// TwinCAT 3 PLC project Untitled1
// ProgramVersion: 3.1.4022.7
// libraries:
//   Tc2_Standard, * (Beckhoff Automation GmbH)
//   Tc2_System, * (Beckhoff Automation GmbH)
//   Tc3_Module, * (Beckhoff Automation GmbH)
// project tree:
//   / PlcTask.TcTTO
//   POUs/ alg_s_Dinitialized.TcPOU, alg_s_Hinitialized.TcPOU, alg_a_Dstartled.TcPOU (not stored), alg_a_Dresetled.TcPOU (not stored), alg_a_DledQ1.TcPOU (not stored), alg_a_DledQ2.TcPOU (not stored), alg_a_pusher1.TcPOU (not stored), alg_a_pusher2.TcPOU (not stored), alg_a_pusher3.TcPOU (not stored), alg_a_Hstartled.TcPOU (not stored), alg_a_Hresetled.TcPOU (not stored), alg_a_HledQ1.TcPOU (not stored), alg_a_HledQ2.TcPOU (not stored), alg_a_x2distributing.TcPOU (not stored), alg_a_x2testing.TcPOU (not stored), alg_a_zdown.TcPOU (not stored), alg_a_gripperclose.TcPOU (not stored), alg_a_transfer2pickpos.TcPOU (not stored), alg_a_transfer2droppos.TcPOU (not stored), alg_a_vacuum.TcPOU (not stored), alg_a_ejectpulse.TcPOU (not stored), alg_a_handlingready.TcPOU (not stored), alg_M_Distributing_a_Dstopled.TcPOU (not stored), alg_M_Distributing_a_Dstartled.TcPOU (not stored), alg_M_Distributing_a_Dresetled.TcPOU (not stored), alg_M_Distributing_pickpos.TcPOU (not stored), makeArray0.TcPOU (not stored), alg_M_Distributing_atpos.TcPOU (not stored), makeArray1.TcPOU (not stored), derivcvar_M_Distributing_t.TcPOU (not stored), ifExprFunc1.TcPOU (not stored), derivcvar_M_HardwareMap_t.TcPOU, MAIN.TcPOU, projArray0.TcPOU (not stored), normProjIdx.TcPOU (not stored), projArray1.TcPOU (not stored)
//   DUTs/ STATE.TcDUT, enum_E.TcDUT
//   GVLs/ INPUTS.TcGVL, TIMERS.TcGVL
// real-time tasks:
//   TASK PlcTask: cycle T#10ms, priority 20, ADS port 350
// I/O:
//   DEVICE Device 2 (EtherCAT), AmsNetId 192.168.1.11.3.1
//     Term 1 (EK1100) [EK1100 EtherCAT Coupler (2A E-Bus)]
//       Term 2 (EL2828) [EL2828 8Ch. Dig. Output 24V, 2A]
//       Term 3 (EL1008) [EL1008 8Ch. Dig. Input 24V, 3ms]
//       Term 4 (EL2024) [EL2024 4Ch. Dig. Output 24V, 2A]
//       Term 5 (EL1008) [EL1008 8Ch. Dig. Input 24V, 3ms]
//       Term 6 (EL2024) [EL2024 4Ch. Dig. Output 24V, 2A]
//       Term 7 (EL1008) [EL1008 8Ch. Dig. Input 24V, 3ms]
//       Term 16 (EL9011) [EL9011 End Terminal]
//     Term 8 (EK1100) [EK1100 EtherCAT Coupler (2A E-Bus)]
//       Term 9 (EL2828) [EL2828 8Ch. Dig. Output 24V, 2A]
//       Term 10 (EL1008) [EL1008 8Ch. Dig. Input 24V, 3ms]
//       Term 11 (EL2024) [EL2024 4Ch. Dig. Output 24V, 2A]
//       Term 12 (EL2024) [EL2024 4Ch. Dig. Output 24V, 2A]
//       Term 13 (EL1008) [EL1008 8Ch. Dig. Input 24V, 3ms]
//       Term 14 (EL2004) [EL2004 4Ch. Dig. Output 24V, 0.5A]
//       Term 15 (EL1008) [EL1008 8Ch. Dig. Input 24V, 3ms]
//       Term 17 (EL9011) [EL9011 End Terminal]
// variable links:
//   Untitled1/Untitled1 Instance <-> Device 2 (EtherCAT)/Term 1 (EK1100)/Term 2 (EL2828)
//     PlcTask Outputs/MAIN.state0.dvar_M_HardwareMap_out_a_DledQ1 <-> Channel 3/Output
//     PlcTask Outputs/MAIN.state0.dvar_M_HardwareMap_out_a_DledQ2 <-> Channel 4/Output
//     PlcTask Outputs/MAIN.state0.dvar_M_HardwareMap_out_a_Dout{4..7} <-> Channel {5..8}/Output  (4 links)
//     PlcTask Outputs/MAIN.state0.dvar_M_HardwareMap_out_a_Dresetled <-> Channel 2/Output
//     PlcTask Outputs/MAIN.state0.dvar_M_HardwareMap_out_a_Dstartled <-> Channel 1/Output
//   Untitled1/Untitled1 Instance <-> Device 2 (EtherCAT)/Term 1 (EK1100)/Term 3 (EL1008)
//     PlcTask Inputs/INPUTS.ivar_s_Dautoswitch <-> Channel 3/Input
//     PlcTask Inputs/INPUTS.ivar_s_Din{4..7} <-> Channel {5..8}/Input  (4 links)
//     PlcTask Inputs/INPUTS.ivar_s_Dresetbutton <-> Channel 4/Input
//     PlcTask Inputs/INPUTS.ivar_s_Dstartbutton <-> Channel 1/Input
//     PlcTask Inputs/INPUTS.ivar_s_Dstopbutton <-> Channel 2/Input
//   Untitled1/Untitled1 Instance <-> Device 2 (EtherCAT)/Term 1 (EK1100)/Term 4 (EL2024)
//     PlcTask Outputs/MAIN.state0.dvar_M_HardwareMap_out_a_pusher1 <-> Channel 1/Output
//     PlcTask Outputs/MAIN.state0.dvar_M_HardwareMap_out_a_pusher2 <-> Channel 2/Output
//     PlcTask Outputs/MAIN.state0.dvar_M_HardwareMap_out_a_pusher3 <-> Channel 3/Output
//   Untitled1/Untitled1 Instance <-> Device 2 (EtherCAT)/Term 1 (EK1100)/Term 5 (EL1008)
//     PlcTask Inputs/INPUTS.ivar_s_product1 <-> Channel 4/Input
//     PlcTask Inputs/INPUTS.ivar_s_product2 <-> Channel 8/Input
//     PlcTask Inputs/INPUTS.ivar_s_pusher1_in <-> Channel 1/Input
//     PlcTask Inputs/INPUTS.ivar_s_pusher2_in <-> Channel 5/Input
//     PlcTask Inputs/INPUTS.ivar_s_pusher1_out <-> Channel 2/Input
//     PlcTask Inputs/INPUTS.ivar_s_pusher2_out <-> Channel 6/Input
//     PlcTask Inputs/INPUTS.ivar_s_stack1filled <-> Channel 3/Input
//     PlcTask Inputs/INPUTS.ivar_s_stack2filled <-> Channel 7/Input
//   Untitled1/Untitled1 Instance <-> Device 2 (EtherCAT)/Term 1 (EK1100)/Term 7 (EL1008)
//     PlcTask Inputs/INPUTS.ivar_s_handlingbusy <-> Channel 8/Input
//     PlcTask Inputs/INPUTS.ivar_s_product3 <-> Channel 4/Input
//     PlcTask Inputs/INPUTS.ivar_s_pusher3_in <-> Channel 1/Input
//     PlcTask Inputs/INPUTS.ivar_s_pusher3_out <-> Channel 2/Input
//     PlcTask Inputs/INPUTS.ivar_s_stack3filled <-> Channel 3/Input
//   Untitled1/Untitled1 Instance <-> Device 2 (EtherCAT)/Term 8 (EK1100)/Term 10 (EL1008)
//     PlcTask Inputs/INPUTS.ivar_s_Hautoswitch <-> Channel 3/Input
//     PlcTask Inputs/INPUTS.ivar_s_Hin{4..7} <-> Channel {5..8}/Input  (4 links)
//     PlcTask Inputs/INPUTS.ivar_s_Hresetbutton <-> Channel 4/Input
//     PlcTask Inputs/INPUTS.ivar_s_Hstartbutton <-> Channel 1/Input
//     PlcTask Inputs/INPUTS.ivar_s_Hstopbutton <-> Channel 2/Input
//   Untitled1/Untitled1 Instance <-> Device 2 (EtherCAT)/Term 8 (EK1100)/Term 11 (EL2024)
//     PlcTask Outputs/MAIN.state0.dvar_M_HardwareMap_out_a_gripperclose <-> Channel 4/Output
//     PlcTask Outputs/MAIN.state0.dvar_M_HardwareMap_out_a_x2distributing <-> Channel 1/Output
//     PlcTask Outputs/MAIN.state0.dvar_M_HardwareMap_out_a_x2testing <-> Channel 2/Output
//     PlcTask Outputs/MAIN.state0.dvar_M_HardwareMap_out_a_zdown <-> Channel 3/Output
//   Untitled1/Untitled1 Instance <-> Device 2 (EtherCAT)/Term 8 (EK1100)/Term 12 (EL2024)
//     PlcTask Outputs/MAIN.state0.dvar_M_HardwareMap_out_a_ejectpulse <-> Channel 4/Output
//     PlcTask Outputs/MAIN.state0.dvar_M_HardwareMap_out_a_transfer2droppos <-> Channel 2/Output
//     PlcTask Outputs/MAIN.state0.dvar_M_HardwareMap_out_a_transfer2pickpos <-> Channel 1/Output
//     PlcTask Outputs/MAIN.state0.dvar_M_HardwareMap_out_a_vacuum <-> Channel 3/Output
//   Untitled1/Untitled1 Instance <-> Device 2 (EtherCAT)/Term 8 (EK1100)/Term 13 (EL1008)
//     PlcTask Inputs/INPUTS.ivar_s_xpos_at1 <-> Channel 4/Input
//     PlcTask Inputs/INPUTS.ivar_s_xpos_at2 <-> Channel 5/Input
//     PlcTask Inputs/INPUTS.ivar_s_xpos_at3 <-> Channel 6/Input
//     PlcTask Inputs/INPUTS.ivar_s_xpos_atdrop <-> Channel 7/Input
//     PlcTask Inputs/INPUTS.ivar_s_zpos_atup <-> Channel 8/Input
//   Untitled1/Untitled1 Instance <-> Device 2 (EtherCAT)/Term 8 (EK1100)/Term 14 (EL2004)
//     PlcTask Outputs/MAIN.state0.dvar_M_HardwareMap_out_a_handlingready <-> Channel 4/Output
//   Untitled1/Untitled1 Instance <-> Device 2 (EtherCAT)/Term 8 (EK1100)/Term 15 (EL1008)
//     PlcTask Inputs/INPUTS.ivar_s_gripper <-> Channel 2/Input
//     PlcTask Inputs/INPUTS.ivar_s_product4 <-> Channel 7/Input
//     PlcTask Inputs/INPUTS.ivar_s_testingbusy <-> Channel 8/Input
//     PlcTask Inputs/INPUTS.ivar_s_transfer_atdrop <-> Channel 4/Input
//     PlcTask Inputs/INPUTS.ivar_s_transfer_athalfway <-> Channel 5/Input
//     PlcTask Inputs/INPUTS.ivar_s_transfer_atpickup <-> Channel 3/Input
//     PlcTask Inputs/INPUTS.ivar_s_vacuum <-> Channel 6/Input
//     PlcTask Inputs/INPUTS.ivar_s_zpos_atdown <-> Channel 1/Input
//   Untitled1/Untitled1 Instance <-> Device 2 (EtherCAT)/Term 8 (EK1100)/Term 9 (EL2828)
//     PlcTask Outputs/MAIN.state0.dvar_M_HardwareMap_out_a_HledQ1 <-> Channel 3/Output
//     PlcTask Outputs/MAIN.state0.dvar_M_HardwareMap_out_a_HledQ2 <-> Channel 4/Output
//     PlcTask Outputs/MAIN.state0.dvar_M_HardwareMap_out_a_Hout{4..7} <-> Channel {5..8}/Output  (4 links)
//     PlcTask Outputs/MAIN.state0.dvar_M_HardwareMap_out_a_Hresetled <-> Channel 2/Output
//     PlcTask Outputs/MAIN.state0.dvar_M_HardwareMap_out_a_Hstartled <-> Channel 1/Output

CONFIGURATION Untitled1
    RESOURCE PLC ON TwinCAT3
        TASK PlcTask(INTERVAL := T#10ms, PRIORITY := 20);
        PROGRAM MAIN WITH PlcTask : MAIN;
    END_RESOURCE
END_CONFIGURATION

// ---- DUTs/STATE.TcDUT
TYPE STATE:
    STRUCT
        curTime: LREAL;
        dvar_M_Distributing_a_x2distributing AT %Q*: BOOL;
        dvar_M_Distributing_a_zdown AT %Q*: BOOL;
        dvar_M_Distributing_a_gripperclose AT %Q*: BOOL;
        dvar_M_Distributing_a_x2testing AT %Q*: BOOL;
        dvar_M_Distributing_i AT %Q*: DINT;
        cvar_M_Distributing_t AT %Q*: LREAL;
        dvar_M_Distributing AT %Q*: enum_E;
        dvar_M_HardwareMap_out_a_Dstartled AT %Q*: BOOL;
        dvar_M_HardwareMap_out_a_Dresetled AT %Q*: BOOL;
        dvar_M_HardwareMap_out_a_DledQ1 AT %Q*: BOOL;
        dvar_M_HardwareMap_out_a_DledQ2 AT %Q*: BOOL;
        dvar_M_HardwareMap_out_a_Dout4 AT %Q*: BOOL;
        dvar_M_HardwareMap_out_a_Dout5 AT %Q*: BOOL;
        dvar_M_HardwareMap_out_a_Dout6 AT %Q*: BOOL;
        dvar_M_HardwareMap_out_a_Dout7 AT %Q*: BOOL;
        dvar_M_HardwareMap_out_a_pusher1 AT %Q*: BOOL;
        dvar_M_HardwareMap_out_a_pusher2 AT %Q*: BOOL;
        dvar_M_HardwareMap_out_a_pusher3 AT %Q*: BOOL;
        dvar_M_HardwareMap_out_a_Hstartled AT %Q*: BOOL;
        dvar_M_HardwareMap_out_a_Hresetled AT %Q*: BOOL;
        dvar_M_HardwareMap_out_a_HledQ1 AT %Q*: BOOL;
        dvar_M_HardwareMap_out_a_HledQ2 AT %Q*: BOOL;
        dvar_M_HardwareMap_out_a_Hout4 AT %Q*: BOOL;
        dvar_M_HardwareMap_out_a_Hout5 AT %Q*: BOOL;
        dvar_M_HardwareMap_out_a_Hout6 AT %Q*: BOOL;
        dvar_M_HardwareMap_out_a_Hout7 AT %Q*: BOOL;
        dvar_M_HardwareMap_out_a_x2distributing AT %Q*: BOOL;
        dvar_M_HardwareMap_out_a_x2testing AT %Q*: BOOL;
        dvar_M_HardwareMap_out_a_zdown AT %Q*: BOOL;
        dvar_M_HardwareMap_out_a_gripperclose AT %Q*: BOOL;
        dvar_M_HardwareMap_out_a_transfer2pickpos AT %Q*: BOOL;
        dvar_M_HardwareMap_out_a_transfer2droppos AT %Q*: BOOL;
        dvar_M_HardwareMap_out_a_vacuum AT %Q*: BOOL;
        dvar_M_HardwareMap_out_a_ejectpulse AT %Q*: BOOL;
        dvar_M_HardwareMap_out_a_handlingready AT %Q*: BOOL;
        dvar_M_HardwareMap_init_err_sen_idx AT %Q*: DINT;
        dvar_M_HardwareMap_init_err_led_idx AT %Q*: DINT;
        cvar_M_HardwareMap_t AT %Q*: LREAL;
        dvar_M_HardwareMap AT %Q*: enum_E;
        dvar_M_inventory1_a_pusher1 AT %Q*: BOOL;
        dvar_M_inventory1 AT %Q*: enum_E;
        dvar_M_inventory2_a_pusher2 AT %Q*: BOOL;
        dvar_M_inventory2 AT %Q*: enum_E;
        dvar_M_inventory3_a_pusher3 AT %Q*: BOOL;
        dvar_M_inventory3 AT %Q*: enum_E;
        dvar_M_vacuum_a_transfer2pickpos AT %Q*: BOOL;
        dvar_M_vacuum_a_transfer2droppos AT %Q*: BOOL;
        dvar_M_vacuum_a_vacuum AT %Q*: BOOL;
        dvar_M_vacuum_a_ejectpulse AT %Q*: BOOL;
        dvar_M_vacuum AT %Q*: enum_E;
    END_STRUCT
END_TYPE

// ---- DUTs/enum_E.TcDUT
TYPE enum_E:
    (elit_clear_vacuum, elit_down, elit_droppoint, elit_finished, elit_goback, elit_going, elit_gopickup, elit_goup, elit_init0, elit_init1, elit_init2, elit_init3, elit_init4, elit_init5, elit_init6, elit_init7, elit_init8, elit_init9, elit_init_error, elit_init_ok, elit_init_sensor_check, elit_initialized, elit_key, elit_movetopickup, elit_pauze_left, elit_pickupvac, elit_reset, elit_reset_button, elit_reset_down, elit_reset_place, elit_rest, elit_starting, elit_stop, elit_testingdrop, elit_wait_start, elit_wait_vacuum);
END_TYPE

// ---- GVLs/INPUTS.TcGVL
VAR_GLOBAL // INPUTS
    ivar_s_Dstartbutton AT %I*: BOOL;
    ivar_s_Dstopbutton AT %I*: BOOL;
    ivar_s_Dresetbutton AT %I*: BOOL;
    ivar_s_Dautoswitch AT %I*: BOOL;
    ivar_s_pusher1_in AT %I*: BOOL;
    ivar_s_pusher1_out AT %I*: BOOL;
    ivar_s_stack1filled AT %I*: BOOL;
    ivar_s_product1 AT %I*: BOOL;
    ivar_s_pusher2_in AT %I*: BOOL;
    ivar_s_pusher2_out AT %I*: BOOL;
    ivar_s_stack2filled AT %I*: BOOL;
    ivar_s_product2 AT %I*: BOOL;
    ivar_s_pusher3_in AT %I*: BOOL;
    ivar_s_pusher3_out AT %I*: BOOL;
    ivar_s_stack3filled AT %I*: BOOL;
    ivar_s_product3 AT %I*: BOOL;
    ivar_s_handlingbusy AT %I*: BOOL;
    ivar_s_Hstartbutton AT %I*: BOOL;
    ivar_s_Hstopbutton AT %I*: BOOL;
    ivar_s_Hresetbutton AT %I*: BOOL;
    ivar_s_Hautoswitch AT %I*: BOOL;
    ivar_s_xpos_at1 AT %I*: BOOL;
    ivar_s_xpos_at2 AT %I*: BOOL;
    ivar_s_xpos_at3 AT %I*: BOOL;
    ivar_s_xpos_atdrop AT %I*: BOOL;
    ivar_s_zpos_atup AT %I*: BOOL;
    ivar_s_zpos_atdown AT %I*: BOOL;
    ivar_s_gripper AT %I*: BOOL;
    ivar_s_transfer_atpickup AT %I*: BOOL;
    ivar_s_transfer_atdrop AT %I*: BOOL;
    ivar_s_transfer_athalfway AT %I*: BOOL;
    ivar_s_vacuum AT %I*: BOOL;
    ivar_s_product4 AT %I*: BOOL;
    ivar_s_testingbusy AT %I*: BOOL;
    ivar_s_Din4 AT %I*: BOOL;
    ivar_s_Din5 AT %I*: BOOL;
    ivar_s_Din6 AT %I*: BOOL;
    ivar_s_Din7 AT %I*: BOOL;
    ivar_s_Hin4 AT %I*: BOOL;
    ivar_s_Hin5 AT %I*: BOOL;
    ivar_s_Hin6 AT %I*: BOOL;
    ivar_s_Hin7 AT %I*: BOOL;
    ivar_a_Dout4 AT %I*: BOOL;
    ivar_a_Dout5 AT %I*: BOOL;
    ivar_a_Dout6 AT %I*: BOOL;
    ivar_a_Dout7 AT %I*: BOOL;
    ivar_a_Hout4 AT %I*: BOOL;
    ivar_a_Hout5 AT %I*: BOOL;
    ivar_a_Hout6 AT %I*: BOOL;
    ivar_a_Hout7 AT %I*: BOOL;
END_VAR

// ---- GVLs/TIMERS.TcGVL
VAR_GLOBAL // TIMERS
    timer0: TON;
    timer1: TON;
    curTimer: INT := 0;
END_VAR

// ---- POUs/MAIN.TcPOU
PROGRAM MAIN
VAR_OUTPUT
    timerValue0: TIME;
    timerValue1: TIME;
END_VAR
VAR
    cnt: LINT;
    first: BOOL := TRUE;
    curTimerValue: TIME;
    state0: STATE;
    curTime: LREAL;
    loopsKilled: LINT;
END_VAR
VAR_TEMP
    lastTimerValue: TIME;
    curDeltaTime: TIME;
    curDeltaSecs: LREAL;
    state1: STATE;
    progress: BOOL;
    loopCount: INT;
    b1: BOOL;
    b2: BOOL;
END_VAR


// Handle 'time' and cycle time.
cnt := cnt + 1;

timer0(IN := curTimer = 0, PT := T#1D);
timer1(IN := curTimer = 1, PT := T#1D);
timerValue0 := timer0.ET;
timerValue1 := timer1.ET;

lastTimerValue := curTimerValue;
IF curTimer = 0 THEN
    curTimerValue := timerValue0;
ELSE
    curTimerValue := timerValue1;
END_IF;
curDeltaTime := curTimerValue - lastTimerValue;
curDeltaSecs := TIME_TO_LREAL(curDeltaTime) / 1000;
curTime := curTime + curDeltaSecs;

IF cnt MOD 10 = 0 THEN
    curTimer := 1 - curTimer;
    curTimerValue := T#0S;
    timer0(IN := curTimer = 0, PT := T#1D);
    timer1(IN := curTimer = 1, PT := T#1D);
    timerValue0 := timer0.ET;
    timerValue1 := timer1.ET;
END_IF;

IF first THEN
    first := FALSE;

    // Initialize state variables for initial state.
    state0.dvar_M_Distributing_a_x2distributing := FALSE;
    state0.dvar_M_Distributing_a_zdown := FALSE;
    state0.dvar_M_Distributing_a_gripperclose := FALSE;
    state0.dvar_M_Distributing_a_x2testing := FALSE;
    state0.dvar_M_Distributing_i := 0;
    state0.cvar_M_Distributing_t := 0.0;
    state0.dvar_M_Distributing := elit_init2;
    state0.dvar_M_HardwareMap_out_a_Dstartled := FALSE;
    state0.dvar_M_HardwareMap_out_a_Dresetled := FALSE;
    state0.dvar_M_HardwareMap_out_a_DledQ1 := TRUE;
    state0.dvar_M_HardwareMap_out_a_DledQ2 := TRUE;
    state0.dvar_M_HardwareMap_out_a_Dout4 := FALSE;
    state0.dvar_M_HardwareMap_out_a_Dout5 := FALSE;
    state0.dvar_M_HardwareMap_out_a_Dout6 := FALSE;
    state0.dvar_M_HardwareMap_out_a_Dout7 := FALSE;
    state0.dvar_M_HardwareMap_out_a_pusher1 := FALSE;
    state0.dvar_M_HardwareMap_out_a_pusher2 := FALSE;
    state0.dvar_M_HardwareMap_out_a_pusher3 := FALSE;
    state0.dvar_M_HardwareMap_out_a_Hstartled := FALSE;
    state0.dvar_M_HardwareMap_out_a_Hresetled := FALSE;
    state0.dvar_M_HardwareMap_out_a_HledQ1 := TRUE;
    state0.dvar_M_HardwareMap_out_a_HledQ2 := TRUE;
    state0.dvar_M_HardwareMap_out_a_Hout4 := FALSE;
    state0.dvar_M_HardwareMap_out_a_Hout5 := FALSE;
    state0.dvar_M_HardwareMap_out_a_Hout6 := FALSE;
    state0.dvar_M_HardwareMap_out_a_Hout7 := FALSE;
    state0.dvar_M_HardwareMap_out_a_x2distributing := TRUE;
    state0.dvar_M_HardwareMap_out_a_x2testing := TRUE;
    state0.dvar_M_HardwareMap_out_a_zdown := FALSE;
    state0.dvar_M_HardwareMap_out_a_gripperclose := FALSE;
    state0.dvar_M_HardwareMap_out_a_transfer2pickpos := FALSE;
    state0.dvar_M_HardwareMap_out_a_transfer2droppos := FALSE;
    state0.dvar_M_HardwareMap_out_a_vacuum := FALSE;
    state0.dvar_M_HardwareMap_out_a_ejectpulse := FALSE;
    state0.dvar_M_HardwareMap_out_a_handlingready := FALSE;
    state0.dvar_M_HardwareMap_init_err_sen_idx := -1;
    state0.dvar_M_HardwareMap_init_err_led_idx := 0;
    state0.cvar_M_HardwareMap_t := 0.0;
    state0.dvar_M_HardwareMap := elit_init0;
    state0.dvar_M_inventory1_a_pusher1 := FALSE;
    state0.dvar_M_inventory1 := elit_init2;
    state0.dvar_M_inventory2_a_pusher2 := FALSE;
    state0.dvar_M_inventory2 := elit_init2;
    state0.dvar_M_inventory3_a_pusher3 := FALSE;
    state0.dvar_M_inventory3 := elit_init2;
    state0.dvar_M_vacuum_a_transfer2pickpos := FALSE;
    state0.dvar_M_vacuum_a_transfer2droppos := FALSE;
    state0.dvar_M_vacuum_a_vacuum := FALSE;
    state0.dvar_M_vacuum_a_ejectpulse := FALSE;
    state0.dvar_M_vacuum := elit_init2;
ELSE
    // Update continuous variables for time delay.
    state1.cvar_M_Distributing_t := state0.cvar_M_Distributing_t + curDeltaSecs * derivcvar_M_Distributing_t(state0);
    state1.cvar_M_HardwareMap_t := state0.cvar_M_HardwareMap_t + curDeltaSecs * derivcvar_M_HardwareMap_t(state0);

    state0.curTime := curTime;
    state0.cvar_M_Distributing_t := state1.cvar_M_Distributing_t;
    state0.cvar_M_HardwareMap_t := state1.cvar_M_HardwareMap_t;
END_IF;

// Event loop.
WHILE TRUE DO
    progress := FALSE;

    // Event "M.inventory1_a".
    IF NOT progress THEN
        b1 := (state0.dvar_M_inventory1) = (elit_starting);
        b1 := b1 AND (ivar_s_pusher1_in);
        b1 := b1 AND (NOT(ivar_s_product1));
        IF b1 THEN
            progress := TRUE;
            state1 := state0;

            state1.dvar_M_inventory1_a_pusher1 := TRUE;
            state1.dvar_M_inventory1 := elit_going;

            state0 := state1;
        END_IF;
    END_IF;

    // Event "M.inventory1_b".
    IF NOT progress THEN
        b1 := (state0.dvar_M_inventory1) = (elit_starting);
        b1 := b1 AND (ivar_s_pusher1_out);
        b1 := b1 AND (ivar_s_stack1filled);
        b1 := b1 AND (state0.dvar_M_inventory1_a_pusher1);
        IF b1 THEN
            progress := TRUE;
            state1 := state0;

            state1.dvar_M_inventory1 := elit_going;

            state0 := state1;
        END_IF;
    END_IF;

    // Event "M.inventory1_c".
    IF NOT progress THEN
        b1 := (state0.dvar_M_inventory1) = (elit_starting);
        b1 := b1 AND (NOT(ivar_s_Dstopbutton));
        IF b1 THEN
            progress := TRUE;
            state1 := state0;

            state1.dvar_M_inventory1_a_pusher1 := FALSE;
            state1.dvar_M_inventory1 := elit_stop;

            state0 := state1;
        END_IF;
    END_IF;

    // Event "M.inventory1_d".
    IF NOT progress THEN
        b1 := (state0.dvar_M_inventory1) = (elit_going);
        b1 := b1 AND (ivar_s_pusher1_out);
        b1 := b1 AND (ivar_s_stack1filled);
        IF b1 THEN
            progress := TRUE;
            state1 := state0;

            state1.dvar_M_inventory1_a_pusher1 := FALSE;
            state1.dvar_M_inventory1 := elit_starting;

            state0 := state1;
        END_IF;
    END_IF;

    // Event "tau".
    IF NOT progress THEN
        b1 := (state0.dvar_M_Distributing) = (elit_init2);
        b1 := b1 AND (alg_s_Dinitialized(state0));
        IF b1 THEN
            progress := TRUE;
            state1 := state0;

            state1.dvar_M_Distributing := elit_wait_start;

            state0 := state1;
        END_IF;
    END_IF;

    // Event "tau".
    IF NOT progress THEN
        b1 := (state0.dvar_M_Distributing) = (elit_wait_start);
        b1 := b1 AND (ivar_s_Dstartbutton);
        IF b1 THEN
            progress := TRUE;
            state1 := state0;

            state1.dvar_M_Distributing := elit_droppoint;

            state0 := state1;
        END_IF;
    END_IF;

    // Event "tau".
    IF NOT progress THEN
        b1 := (state0.dvar_M_Distributing) = (elit_reset_button);
        b1 := b1 AND (NOT(ivar_s_Dstopbutton));
        IF b1 THEN
            progress := TRUE;
            state1 := state0;

            state1.dvar_M_Distributing_a_x2distributing := FALSE;
            state1.dvar_M_Distributing_a_x2testing := FALSE;
            state1.dvar_M_Distributing_a_zdown := FALSE;
            state1.dvar_M_Distributing := elit_stop;

            state0 := state1;
        END_IF;
    END_IF;

    // Event "tau".
    IF NOT progress THEN
        b1 := (state0.dvar_M_Distributing) = (elit_reset_button);
        b1 := b1 AND (ivar_s_gripper);
        b1 := b1 AND (ivar_s_xpos_at3);
        IF b1 THEN
            progress := TRUE;
            state1 := state0;

            state1.dvar_M_Distributing_a_zdown := FALSE;
            state1.dvar_M_Distributing_a_x2distributing := TRUE;
            state1.dvar_M_Distributing := elit_wait_vacuum;

            state0 := state1;
        END_IF;
    END_IF;

    // Event "tau".
    IF NOT progress THEN
        b1 := (state0.dvar_M_Distributing) = (elit_reset_button);
        b1 := b1 AND (ivar_s_gripper);
        b1 := b1 AND (ivar_s_xpos_atdrop);
        IF b1 THEN
            progress := TRUE;
            state1 := state0;

            state1.dvar_M_Distributing_a_zdown := FALSE;
            state1.dvar_M_Distributing_a_x2distributing := TRUE;
            state1.dvar_M_Distributing_a_x2testing := FALSE;
            state1.dvar_M_Distributing := elit_pauze_left;

            state0 := state1;
        END_IF;
    END_IF;

    // Event "tau".
    IF NOT progress THEN
        b1 := (state0.dvar_M_Distributing) = (elit_reset_button);
        b1 := b1 AND (NOT(ivar_s_gripper));
        b1 := b1 AND (ivar_s_xpos_at3);
        IF b1 THEN
            progress := TRUE;
            state1 := state0;

            state1.dvar_M_Distributing_a_zdown := FALSE;
            state1.dvar_M_Distributing_a_x2distributing := TRUE;
            state1.dvar_M_Distributing := elit_wait_vacuum;

            state0 := state1;
        END_IF;
    END_IF;

    // Event "tau".
    IF NOT progress THEN
        b1 := (state0.dvar_M_Distributing) = (elit_reset_button);
        b1 := b1 AND (NOT(ivar_s_gripper));
        b1 := b1 AND (ivar_s_xpos_atdrop);
        IF b1 THEN
            progress := TRUE;
            state1 := state0;

            state1.dvar_M_Distributing_a_zdown := FALSE;
            state1.dvar_M_Distributing_a_x2distributing := TRUE;
            state1.dvar_M_Distributing_a_x2testing := FALSE;
            state1.dvar_M_Distributing := elit_pauze_left;

            state0 := state1;
        END_IF;
    END_IF;

    // Event "tau".
    IF NOT progress THEN
        b1 := (state0.dvar_M_Distributing) = (elit_pauze_left);
        b1 := b1 AND (NOT(ivar_s_Dstopbutton));
        IF b1 THEN
            progress := TRUE;
            state1 := state0;

            state1.dvar_M_Distributing_a_x2distributing := FALSE;
            state1.dvar_M_Distributing_a_x2testing := FALSE;
            state1.dvar_M_Distributing_a_zdown := FALSE;
            state1.dvar_M_Distributing := elit_stop;

            state0 := state1;
        END_IF;
    END_IF;

    // Event "tau".
    IF NOT progress THEN
        b1 := (state0.dvar_M_Distributing) = (elit_pauze_left);
        b1 := b1 AND (NOT(ivar_s_gripper));
        b1 := b1 AND (ivar_s_xpos_at3);
        IF b1 THEN
            progress := TRUE;
            state1 := state0;

            state1.dvar_M_Distributing_a_zdown := FALSE;
            state1.dvar_M_Distributing_a_x2distributing := TRUE;
            state1.dvar_M_Distributing_a_x2testing := TRUE;
            state1.dvar_M_Distributing := elit_wait_vacuum;

            state0 := state1;
        END_IF;
    END_IF;

    // Event "tau".
    IF NOT progress THEN
        b1 := (state0.dvar_M_Distributing) = (elit_pauze_left);
        b1 := b1 AND (ivar_s_gripper);
        b1 := b1 AND (ivar_s_xpos_at3);
        IF b1 THEN
            progress := TRUE;
            state1 := state0;

            state1.dvar_M_Distributing_a_zdown := FALSE;
            state1.dvar_M_Distributing_a_x2distributing := TRUE;
            state1.dvar_M_Distributing_a_x2testing := TRUE;
            state1.dvar_M_Distributing := elit_wait_vacuum;

            state0 := state1;
        END_IF;
    END_IF;

    // Event "tau".
    IF NOT progress THEN
        b1 := (state0.dvar_M_Distributing) = (elit_wait_vacuum);
        b1 := b1 AND (NOT(ivar_s_Dstopbutton));
        IF b1 THEN
            progress := TRUE;
            state1 := state0;

            state1.dvar_M_Distributing_a_x2distributing := FALSE;
            state1.dvar_M_Distributing_a_x2testing := FALSE;
            state1.dvar_M_Distributing_a_zdown := FALSE;
            state1.dvar_M_Distributing := elit_stop;

            state0 := state1;
        END_IF;
    END_IF;

    // Event "tau".
    IF NOT progress THEN
        b1 := (state0.dvar_M_Distributing) = (elit_wait_vacuum);
        b1 := b1 AND (NOT(ivar_s_gripper));
        b1 := b1 AND (ivar_s_transfer_athalfway);
        IF b1 THEN
            progress := TRUE;
            state1 := state0;

            state1.dvar_M_Distributing_a_zdown := FALSE;
            state1.dvar_M_Distributing_a_x2distributing := FALSE;
            state1.dvar_M_Distributing_a_x2testing := TRUE;
            state1.dvar_M_Distributing := elit_finished;

            state0 := state1;
        END_IF;
    END_IF;

    // Event "tau".
    IF NOT progress THEN
        b1 := (state0.dvar_M_Distributing) = (elit_wait_vacuum);
        b1 := b1 AND (ivar_s_gripper);
        b1 := b1 AND (ivar_s_transfer_athalfway);
        IF b1 THEN
            progress := TRUE;
            state1 := state0;

            state1.dvar_M_Distributing_a_zdown := FALSE;
            state1.dvar_M_Distributing_a_x2distributing := FALSE;
            state1.dvar_M_Distributing_a_x2testing := TRUE;
            state1.dvar_M_Distributing := elit_reset_down;

            state0 := state1;
        END_IF;
    END_IF;

    // Event "tau".
    IF NOT progress THEN
        b1 := (state0.dvar_M_Distributing) = (elit_reset_down);
        b1 := b1 AND (NOT(ivar_s_Dstopbutton));
        IF b1 THEN
            progress := TRUE;
            state1 := state0;

            state1.dvar_M_Distributing_a_x2distributing := FALSE;
            state1.dvar_M_Distributing_a_x2testing := FALSE;
            state1.dvar_M_Distributing_a_zdown := FALSE;
            state1.dvar_M_Distributing := elit_stop;

            state0 := state1;
        END_IF;
    END_IF;

    // Event "tau".
    IF NOT progress THEN
        b1 := (state0.dvar_M_Distributing) = (elit_reset_down);
        b1 := b1 AND (ivar_s_xpos_atdrop);
        IF b1 THEN
            progress := TRUE;
            state1 := state0;

            state1.dvar_M_Distributing_a_zdown := TRUE;
            state1.dvar_M_Distributing_a_x2distributing := TRUE;
            state1.dvar_M_Distributing := elit_reset_place;

            state0 := state1;
        END_IF;
    END_IF;

    // Event "tau".
    IF NOT progress THEN
        b1 := (state0.dvar_M_Distributing) = (elit_reset_place);
        b1 := b1 AND (NOT(ivar_s_Dstopbutton));
        IF b1 THEN
            progress := TRUE;
            state1 := state0;

            state1.dvar_M_Distributing_a_x2distributing := FALSE;
            state1.dvar_M_Distributing_a_x2testing := FALSE;
            state1.dvar_M_Distributing_a_zdown := FALSE;
            state1.dvar_M_Distributing := elit_stop;

            state0 := state1;
        END_IF;
    END_IF;

    // Event "tau".
    IF NOT progress THEN
        b1 := (state0.dvar_M_Distributing) = (elit_reset_place);
        b1 := b1 AND (ivar_s_zpos_atdown);
        IF b1 THEN
            progress := TRUE;
            state1 := state0;

            state1.cvar_M_Distributing_t := 0.0;
            state1.dvar_M_Distributing_a_gripperclose := FALSE;
            state1.dvar_M_Distributing_a_zdown := FALSE;
            state1.dvar_M_Distributing_a_x2distributing := FALSE;
            state1.dvar_M_Distributing_a_x2testing := FALSE;
            state1.dvar_M_Distributing := elit_finished;

            state0 := state1;
        END_IF;
    END_IF;

    // Event "tau".
    IF NOT progress THEN
        b1 := (state0.dvar_M_Distributing) = (elit_stop);
        b1 := b1 AND (ivar_s_Dstartbutton);
        IF b1 THEN
            progress := TRUE;
            state1 := state0;

            state1.dvar_M_Distributing_a_x2testing := TRUE;
            state1.dvar_M_Distributing := elit_droppoint;

            state0 := state1;
        END_IF;
    END_IF;

    // Event "tau".
    IF NOT progress THEN
        b1 := (state0.dvar_M_Distributing) = (elit_stop);
        b1 := b1 AND (ivar_s_Dresetbutton);
        IF b1 THEN
            progress := TRUE;
            state1 := state0;

            state1.dvar_M_Distributing_a_x2distributing := FALSE;
            state1.dvar_M_Distributing_a_x2testing := TRUE;
            state1.dvar_M_Distributing := elit_reset_button;

            state0 := state1;
        END_IF;
    END_IF;

    // Event "tau".
    IF NOT progress THEN
        b1 := (state0.dvar_M_Distributing) = (elit_droppoint);
        b1 := b1 AND (ivar_s_Dresetbutton);
        IF b1 THEN
            progress := TRUE;
            state1 := state0;

            state1.dvar_M_Distributing_a_x2distributing := FALSE;
            state1.dvar_M_Distributing_a_x2testing := TRUE;
            state1.dvar_M_Distributing := elit_reset_button;

            state0 := state1;
        END_IF;
    END_IF;

    // Event "tau".
    IF NOT progress THEN
        b1 := (state0.dvar_M_Distributing) = (elit_droppoint);
        b1 := b1 AND (NOT(ivar_s_Dstopbutton));
        IF b1 THEN
            progress := TRUE;
            state1 := state0;

            state1.dvar_M_Distributing_a_x2distributing := FALSE;
            state1.dvar_M_Distributing_a_x2testing := FALSE;
            state1.dvar_M_Distributing_a_zdown := FALSE;
            state1.dvar_M_Distributing := elit_stop;

            state0 := state1;
        END_IF;
    END_IF;

    // Event "tau".
    IF NOT progress THEN
        b1 := (state0.dvar_M_Distributing) = (elit_droppoint);
        b1 := b1 AND (ivar_s_gripper);
        b1 := b1 AND (ivar_s_xpos_atdrop);
        b1 := b1 AND (ivar_s_zpos_atup);
        IF b1 THEN
            progress := TRUE;
            state1 := state0;

            state1.dvar_M_Distributing_a_x2distributing := TRUE;
            state1.dvar_M_Distributing_a_x2testing := TRUE;
            state1.dvar_M_Distributing := elit_down;

            state0 := state1;
        END_IF;
    END_IF;

    // Event "tau".
    IF NOT progress THEN
        b1 := (state0.dvar_M_Distributing) = (elit_droppoint);
        b1 := b1 AND (NOT(ivar_s_gripper));
        b1 := b1 AND (ivar_s_xpos_atdrop);
        b1 := b1 AND (ivar_s_zpos_atup);
        IF b1 THEN
            progress := TRUE;
            state1 := state0;

            state1.dvar_M_Distributing_a_x2distributing := TRUE;
            state1.dvar_M_Distributing_a_x2testing := FALSE;
            state1.dvar_M_Distributing := elit_movetopickup;

            state0 := state1;
        END_IF;
    END_IF;

    // Event "tau".
    IF NOT progress THEN
        b1 := (state0.dvar_M_Distributing) = (elit_movetopickup);
        b1 := b1 AND (ivar_s_Dresetbutton);
        IF b1 THEN
            progress := TRUE;
            state1 := state0;

            state1.dvar_M_Distributing_a_x2distributing := FALSE;
            state1.dvar_M_Distributing_a_x2testing := TRUE;
            state1.dvar_M_Distributing := elit_reset_button;

            state0 := state1;
        END_IF;
    END_IF;

    // Event "tau".
    IF NOT progress THEN
        b1 := (state0.dvar_M_Distributing) = (elit_movetopickup);
        b1 := b1 AND (NOT(ivar_s_Dstopbutton));
        IF b1 THEN
            progress := TRUE;
            state1 := state0;

            state1.dvar_M_Distributing_a_x2distributing := FALSE;
            state1.dvar_M_Distributing_a_x2testing := FALSE;
            state1.dvar_M_Distributing_a_zdown := FALSE;
            state1.dvar_M_Distributing := elit_stop;

            state0 := state1;
        END_IF;
    END_IF;

    // Event "tau".
    IF NOT progress THEN
        b1 := (state0.dvar_M_Distributing) = (elit_movetopickup);
        b1 := b1 AND (projArray1(alg_M_Distributing_atpos(state0), projArray0(makeArray0(0, 1, 0, 2), state0.dvar_M_Distributing_i)));
        b1 := b1 AND ((state0.dvar_M_Distributing_i) < (3));
        IF b1 THEN
            progress := TRUE;
            state1 := state0;

            state1.dvar_M_Distributing_i := (state0.dvar_M_Distributing_i) + (1);
            state1.dvar_M_Distributing_a_x2distributing := TRUE;
            state1.dvar_M_Distributing_a_x2testing := TRUE;
            state1.dvar_M_Distributing := elit_down;

            state0 := state1;
        END_IF;
    END_IF;

    // Event "tau".
    IF NOT progress THEN
        b1 := (state0.dvar_M_Distributing) = (elit_movetopickup);
        b1 := b1 AND (projArray1(alg_M_Distributing_atpos(state0), projArray0(makeArray0(0, 1, 0, 2), state0.dvar_M_Distributing_i)));
        b1 := b1 AND ((state0.dvar_M_Distributing_i) >= (3));
        IF b1 THEN
            progress := TRUE;
            state1 := state0;

            state1.dvar_M_Distributing_i := 0;
            state1.dvar_M_Distributing_a_x2distributing := TRUE;
            state1.dvar_M_Distributing_a_x2testing := TRUE;
            state1.dvar_M_Distributing := elit_down;

            state0 := state1;
        END_IF;
    END_IF;

    // Event "tau".
    IF NOT progress THEN
        b1 := (state0.dvar_M_Distributing) = (elit_down);
        b1 := b1 AND (ivar_s_Dresetbutton);
        IF b1 THEN
            progress := TRUE;
            state1 := state0;

            state1.dvar_M_Distributing_a_x2distributing := FALSE;
            state1.dvar_M_Distributing_a_x2testing := TRUE;
            state1.dvar_M_Distributing := elit_reset_button;

            state0 := state1;
        END_IF;
    END_IF;

    // Event "tau".
    IF NOT progress THEN
        b1 := (state0.dvar_M_Distributing) = (elit_down);
        b1 := b1 AND (NOT(ivar_s_Dstopbutton));
        IF b1 THEN
            progress := TRUE;
            state1 := state0;

            state1.dvar_M_Distributing_a_x2distributing := FALSE;
            state1.dvar_M_Distributing_a_x2testing := FALSE;
            state1.dvar_M_Distributing_a_zdown := FALSE;
            state1.dvar_M_Distributing := elit_stop;

            state0 := state1;
        END_IF;
    END_IF;

    // Event "tau".
    IF NOT progress THEN
        IF (state0.dvar_M_Distributing) = (elit_down) THEN
            progress := TRUE;
            state1 := state0;

            state1.dvar_M_Distributing_a_zdown := TRUE;
            state1.dvar_M_Distributing := elit_gopickup;

            state0 := state1;
        END_IF;
    END_IF;

    // Event "tau".
    IF NOT progress THEN
        b1 := (state0.dvar_M_Distributing) = (elit_gopickup);
        b1 := b1 AND (ivar_s_Dresetbutton);
        IF b1 THEN
            progress := TRUE;
            state1 := state0;

            state1.dvar_M_Distributing_a_x2distributing := FALSE;
            state1.dvar_M_Distributing_a_x2testing := TRUE;
            state1.dvar_M_Distributing := elit_reset_button;

            state0 := state1;
        END_IF;
    END_IF;

    // Event "tau".
    IF NOT progress THEN
        b1 := (state0.dvar_M_Distributing) = (elit_gopickup);
        b1 := b1 AND (NOT(ivar_s_Dstopbutton));
        IF b1 THEN
            progress := TRUE;
            state1 := state0;

            state1.dvar_M_Distributing_a_x2distributing := FALSE;
            state1.dvar_M_Distributing_a_x2testing := FALSE;
            state1.dvar_M_Distributing_a_zdown := FALSE;
            state1.dvar_M_Distributing := elit_stop;

            state0 := state1;
        END_IF;
    END_IF;

    // Event "tau".
    IF NOT progress THEN
        b1 := (state0.dvar_M_Distributing) = (elit_gopickup);
        b1 := b1 AND (ivar_s_zpos_atdown);
        b1 := b1 AND (ivar_s_gripper);
        b1 := b1 AND (NOT(ivar_s_xpos_atdrop));
        IF b1 THEN
            progress := TRUE;
            state1 := state0;

            state1.dvar_M_Distributing_a_gripperclose := TRUE;
            state1.dvar_M_Distributing := elit_goup;

            state0 := state1;
        END_IF;
    END_IF;

    // Event "tau".
    IF NOT progress THEN
        b1 := (state0.dvar_M_Distributing) = (elit_gopickup);
        b1 := b1 AND (ivar_s_zpos_atdown);
        b1 := b1 AND (ivar_s_gripper);
        b1 := b1 AND (ivar_s_xpos_atdrop);
        IF b1 THEN
            progress := TRUE;
            state1 := state0;

            state1.dvar_M_Distributing_a_gripperclose := FALSE;
            state1.dvar_M_Distributing_a_zdown := FALSE;
            state1.dvar_M_Distributing := elit_droppoint;

            state0 := state1;
        END_IF;
    END_IF;

    // Event "tau".
    IF NOT progress THEN
        b1 := (state0.dvar_M_Distributing) = (elit_goup);
        b1 := b1 AND ((state0.cvar_M_Distributing_t) >= (0.1));
        IF b1 THEN
            progress := TRUE;
            state1 := state0;

            state1.cvar_M_Distributing_t := 0.0;
            state1.dvar_M_Distributing_a_zdown := FALSE;
            state1.dvar_M_Distributing := elit_goback;

            state0 := state1;
        END_IF;
    END_IF;

    // Event "tau".
    IF NOT progress THEN
        b1 := (state0.dvar_M_Distributing) = (elit_goback);
        b1 := b1 AND (ivar_s_Dresetbutton);
        IF b1 THEN
            progress := TRUE;
            state1 := state0;

            state1.dvar_M_Distributing_a_x2distributing := FALSE;
            state1.dvar_M_Distributing_a_x2testing := TRUE;
            state1.dvar_M_Distributing := elit_reset_button;

            state0 := state1;
        END_IF;
    END_IF;

    // Event "tau".
    IF NOT progress THEN
        b1 := (state0.dvar_M_Distributing) = (elit_goback);
        b1 := b1 AND (NOT(ivar_s_Dstopbutton));
        IF b1 THEN
            progress := TRUE;
            state1 := state0;

            state1.dvar_M_Distributing_a_x2distributing := FALSE;
            state1.dvar_M_Distributing_a_x2testing := FALSE;
            state1.dvar_M_Distributing_a_zdown := FALSE;
            state1.dvar_M_Distributing := elit_stop;

            state0 := state1;
        END_IF;
    END_IF;

    // Event "tau".
    IF NOT progress THEN
        b1 := (state0.dvar_M_Distributing) = (elit_goback);
        b1 := b1 AND (ivar_s_zpos_atup);
        b1 := b1 AND (ivar_s_gripper);
        b1 := b1 AND ((state0.cvar_M_Distributing_t) > (1));
        IF b1 THEN
            progress := TRUE;
            state1 := state0;

            state1.dvar_M_Distributing_a_x2testing := TRUE;
            state1.dvar_M_Distributing_a_x2distributing := FALSE;
            state1.cvar_M_Distributing_t := 0.0;
            state1.dvar_M_Distributing := elit_droppoint;

            state0 := state1;
        END_IF;
    END_IF;

    // Event "tau".
    IF NOT progress THEN
        b1 := (state0.dvar_M_Distributing) = (elit_finished);
        b1 := b1 AND (NOT(ivar_s_Dstopbutton));
        IF b1 THEN
            progress := TRUE;
            state1 := state0;

            state1.dvar_M_Distributing_a_x2distributing := FALSE;
            state1.dvar_M_Distributing_a_x2testing := FALSE;
            state1.dvar_M_Distributing_a_zdown := FALSE;
            state1.dvar_M_Distributing := elit_stop;

            state0 := state1;
        END_IF;
    END_IF;

    // Event "tau".
    IF NOT progress THEN
        b1 := (state0.dvar_M_Distributing) = (elit_finished);
        b1 := b1 AND (ivar_s_xpos_atdrop);
        IF b1 THEN
            progress := TRUE;
            state1 := state0;

            state1.dvar_M_Distributing_a_x2distributing := TRUE;
            state1.dvar_M_Distributing_a_x2testing := TRUE;
            state1.dvar_M_Distributing := elit_reset;

            state0 := state1;
        END_IF;
    END_IF;

    // Event "tau".
    IF NOT progress THEN
        b1 := (state0.dvar_M_Distributing) = (elit_reset);
        b1 := b1 AND (NOT(ivar_s_Dstopbutton));
        IF b1 THEN
            progress := TRUE;
            state1 := state0;

            state1.dvar_M_Distributing_a_x2distributing := FALSE;
            state1.dvar_M_Distributing_a_x2testing := FALSE;
            state1.dvar_M_Distributing_a_zdown := FALSE;
            state1.dvar_M_Distributing := elit_stop;

            state0 := state1;
        END_IF;
    END_IF;

    // Event "tau".
    IF NOT progress THEN
        b1 := (state0.dvar_M_Distributing) = (elit_reset);
        b1 := b1 AND ((state0.cvar_M_Distributing_t) > (1));
        IF b1 THEN
            progress := TRUE;
            state1 := state0;

            state1.cvar_M_Distributing_t := 0.0;
            state1.dvar_M_Distributing_a_x2distributing := FALSE;
            state1.dvar_M_Distributing_a_x2testing := FALSE;
            state1.dvar_M_Distributing := elit_wait_start;

            state0 := state1;
        END_IF;
    END_IF;

    // Event "tau".
    IF NOT progress THEN
        b1 := (state0.dvar_M_HardwareMap) = (elit_init0);
        b1 := b1 AND ((state0.cvar_M_HardwareMap_t) >= (2.0));
        IF b1 THEN
            progress := TRUE;
            state1 := state0;

            state1.dvar_M_HardwareMap := elit_init1;

            state0 := state1;
        END_IF;
    END_IF;

    // Event "tau".
    IF NOT progress THEN
        IF (state0.dvar_M_HardwareMap) = (elit_init1) THEN
            progress := TRUE;
            state1 := state0;

            state1.dvar_M_HardwareMap_out_a_x2testing := FALSE;
            state1.dvar_M_HardwareMap := elit_init2;

            state0 := state1;
        END_IF;
    END_IF;

    // Event "tau".
    IF NOT progress THEN
        b1 := (state0.dvar_M_HardwareMap) = (elit_init2);
        IF b1 THEN
            b2 := ivar_s_xpos_at1;
            b2 := b2 OR (ivar_s_xpos_at2);
            b1 := b1 AND (b2);
        END_IF;
        IF b1 THEN
            progress := TRUE;
            state1 := state0;

            state1.dvar_M_HardwareMap_out_a_x2testing := TRUE;
            state1.dvar_M_HardwareMap := elit_init3;

            state0 := state1;
        END_IF;
    END_IF;

    // Event "tau".
    IF NOT progress THEN
        IF (state0.dvar_M_HardwareMap) = (elit_init3) THEN
            progress := TRUE;
            state1 := state0;

            state1.dvar_M_HardwareMap_out_a_transfer2pickpos := TRUE;
            state1.dvar_M_HardwareMap := elit_init4;

            state0 := state1;
        END_IF;
    END_IF;

    // Event "tau".
    IF NOT progress THEN
        b1 := (state0.dvar_M_HardwareMap) = (elit_init4);
        b1 := b1 AND (ivar_s_transfer_atpickup);
        IF b1 THEN
            progress := TRUE;
            state1 := state0;

            state1.dvar_M_HardwareMap_out_a_transfer2pickpos := FALSE;
            state1.dvar_M_HardwareMap := elit_init5;

            state0 := state1;
        END_IF;
    END_IF;

    // Event "tau".
    IF NOT progress THEN
        IF (state0.dvar_M_HardwareMap) = (elit_init5) THEN
            progress := TRUE;
            state1 := state0;

            state1.dvar_M_HardwareMap_out_a_transfer2droppos := TRUE;
            state1.dvar_M_HardwareMap := elit_init6;

            state0 := state1;
        END_IF;
    END_IF;

    // Event "tau".
    IF NOT progress THEN
        b1 := (state0.dvar_M_HardwareMap) = (elit_init6);
        b1 := b1 AND (ivar_s_transfer_athalfway);
        IF b1 THEN
            progress := TRUE;
            state1 := state0;

            state1.dvar_M_HardwareMap_out_a_transfer2droppos := FALSE;
            state1.dvar_M_HardwareMap := elit_init7;

            state0 := state1;
        END_IF;
    END_IF;

    // Event "tau".
    IF NOT progress THEN
        IF (state0.dvar_M_HardwareMap) = (elit_init7) THEN
            progress := TRUE;
            state1 := state0;

            state1.dvar_M_HardwareMap_out_a_x2distributing := FALSE;
            state1.dvar_M_HardwareMap := elit_init8;

            state0 := state1;
        END_IF;
    END_IF;

    // Event "tau".
    IF NOT progress THEN
        b1 := (state0.dvar_M_HardwareMap) = (elit_init8);
        b1 := b1 AND (ivar_s_xpos_atdrop);
        IF b1 THEN
            progress := TRUE;
            state1 := state0;

            state1.dvar_M_HardwareMap_out_a_x2distributing := TRUE;
            state1.cvar_M_HardwareMap_t := 0.0;
            state1.dvar_M_HardwareMap := elit_init9;

            state0 := state1;
        END_IF;
    END_IF;

    // Event "tau".
    IF NOT progress THEN
        b1 := (state0.dvar_M_HardwareMap) = (elit_init9);
        b1 := b1 AND ((state0.cvar_M_HardwareMap_t) >= (1));
        IF b1 THEN
            progress := TRUE;
            state1 := state0;

            state1.dvar_M_HardwareMap := elit_init_sensor_check;

            state0 := state1;
        END_IF;
    END_IF;

    // Event "tau".
    IF NOT progress THEN
        b1 := (state0.dvar_M_HardwareMap) = (elit_init_sensor_check);
        b1 := b1 AND (ivar_s_Dstartbutton);
        IF b1 THEN
            progress := TRUE;
            state1 := state0;

            state1.dvar_M_HardwareMap_init_err_sen_idx := 0;
            state1.dvar_M_HardwareMap := elit_init_error;

            state0 := state1;
        END_IF;
    END_IF;

    // Event "tau".
    IF NOT progress THEN
        b1 := (state0.dvar_M_HardwareMap) = (elit_init_sensor_check);
        b1 := b1 AND (NOT(ivar_s_Dstopbutton));
        IF b1 THEN
            progress := TRUE;
            state1 := state0;

            state1.dvar_M_HardwareMap_init_err_sen_idx := 1;
            state1.dvar_M_HardwareMap := elit_init_error;

            state0 := state1;
        END_IF;
    END_IF;

    // Event "tau".
    IF NOT progress THEN
        b1 := (state0.dvar_M_HardwareMap) = (elit_init_sensor_check);
        b1 := b1 AND (ivar_s_Dautoswitch);
        IF b1 THEN
            progress := TRUE;
            state1 := state0;

            state1.dvar_M_HardwareMap_init_err_sen_idx := 2;
            state1.dvar_M_HardwareMap := elit_init_error;

            state0 := state1;
        END_IF;
    END_IF;

    // Event "tau".
    IF NOT progress THEN
        b1 := (state0.dvar_M_HardwareMap) = (elit_init_sensor_check);
        b1 := b1 AND (ivar_s_Dresetbutton);
        IF b1 THEN
            progress := TRUE;
            state1 := state0;

            state1.dvar_M_HardwareMap_init_err_sen_idx := 3;
            state1.dvar_M_HardwareMap := elit_init_error;

            state0 := state1;
        END_IF;
    END_IF;

    // Event "tau".
    IF NOT progress THEN
        b1 := (state0.dvar_M_HardwareMap) = (elit_init_sensor_check);
        b1 := b1 AND (ivar_s_Din4);
        IF b1 THEN
            progress := TRUE;
            state1 := state0;

            state1.dvar_M_HardwareMap_init_err_sen_idx := 4;
            state1.dvar_M_HardwareMap := elit_init_error;

            state0 := state1;
        END_IF;
    END_IF;

    // Event "tau".
    IF NOT progress THEN
        b1 := (state0.dvar_M_HardwareMap) = (elit_init_sensor_check);
        b1 := b1 AND (ivar_s_Din5);
        IF b1 THEN
            progress := TRUE;
            state1 := state0;

            state1.dvar_M_HardwareMap_init_err_sen_idx := 5;
            state1.dvar_M_HardwareMap := elit_init_error;

            state0 := state1;
        END_IF;
    END_IF;

    // Event "tau".
    IF NOT progress THEN
        b1 := (state0.dvar_M_HardwareMap) = (elit_init_sensor_check);
        b1 := b1 AND (ivar_s_Din6);
        IF b1 THEN
            progress := TRUE;
            state1 := state0;

            state1.dvar_M_HardwareMap_init_err_sen_idx := 6;
            state1.dvar_M_HardwareMap := elit_init_error;

            state0 := state1;
        END_IF;
    END_IF;

    // Event "tau".
    IF NOT progress THEN
        b1 := (state0.dvar_M_HardwareMap) = (elit_init_sensor_check);
        b1 := b1 AND (ivar_s_Din7);
        IF b1 THEN
            progress := TRUE;
            state1 := state0;

            state1.dvar_M_HardwareMap_init_err_sen_idx := 7;
            state1.dvar_M_HardwareMap := elit_init_error;

            state0 := state1;
        END_IF;
    END_IF;

    // Event "tau".
    IF NOT progress THEN
        b1 := (state0.dvar_M_HardwareMap) = (elit_init_sensor_check);
        b1 := b1 AND (NOT(ivar_s_pusher1_in));
        IF b1 THEN
            progress := TRUE;
            state1 := state0;

            state1.dvar_M_HardwareMap_init_err_sen_idx := 8;
            state1.dvar_M_HardwareMap := elit_init_error;

            state0 := state1;
        END_IF;
    END_IF;

    // Event "tau".
    IF NOT progress THEN
        b1 := (state0.dvar_M_HardwareMap) = (elit_init_sensor_check);
        b1 := b1 AND (ivar_s_pusher1_out);
        IF b1 THEN
            progress := TRUE;
            state1 := state0;

            state1.dvar_M_HardwareMap_init_err_sen_idx := 9;
            state1.dvar_M_HardwareMap := elit_init_error;

            state0 := state1;
        END_IF;
    END_IF;

    // Event "tau".
    IF NOT progress THEN
        b1 := (state0.dvar_M_HardwareMap) = (elit_init_sensor_check);
        b1 := b1 AND (NOT(ivar_s_stack1filled));
        IF b1 THEN
            progress := TRUE;
            state1 := state0;

            state1.dvar_M_HardwareMap_init_err_sen_idx := 10;
            state1.dvar_M_HardwareMap := elit_init_error;

            state0 := state1;
        END_IF;
    END_IF;

    // Event "tau".
    IF NOT progress THEN
        b1 := (state0.dvar_M_HardwareMap) = (elit_init_sensor_check);
        b1 := b1 AND (ivar_s_product1);
        IF b1 THEN
            progress := TRUE;
            state1 := state0;

            state1.dvar_M_HardwareMap_init_err_sen_idx := 11;
            state1.dvar_M_HardwareMap := elit_init_error;

            state0 := state1;
        END_IF;
    END_IF;

    // Event "tau".
    IF NOT progress THEN
        b1 := (state0.dvar_M_HardwareMap) = (elit_init_sensor_check);
        b1 := b1 AND (NOT(ivar_s_pusher2_in));
        IF b1 THEN
            progress := TRUE;
            state1 := state0;

            state1.dvar_M_HardwareMap_init_err_sen_idx := 12;
            state1.dvar_M_HardwareMap := elit_init_error;

            state0 := state1;
        END_IF;
    END_IF;

    // Event "tau".
    IF NOT progress THEN
        b1 := (state0.dvar_M_HardwareMap) = (elit_init_sensor_check);
        b1 := b1 AND (ivar_s_pusher2_out);
        IF b1 THEN
            progress := TRUE;
            state1 := state0;

            state1.dvar_M_HardwareMap_init_err_sen_idx := 13;
            state1.dvar_M_HardwareMap := elit_init_error;

            state0 := state1;
        END_IF;
    END_IF;

    // Event "tau".
    IF NOT progress THEN
        b1 := (state0.dvar_M_HardwareMap) = (elit_init_sensor_check);
        b1 := b1 AND (NOT(ivar_s_stack2filled));
        IF b1 THEN
            progress := TRUE;
            state1 := state0;

            state1.dvar_M_HardwareMap_init_err_sen_idx := 14;
            state1.dvar_M_HardwareMap := elit_init_error;

            state0 := state1;
        END_IF;
    END_IF;

    // Event "tau".
    IF NOT progress THEN
        b1 := (state0.dvar_M_HardwareMap) = (elit_init_sensor_check);
        b1 := b1 AND (ivar_s_product2);
        IF b1 THEN
            progress := TRUE;
            state1 := state0;

            state1.dvar_M_HardwareMap_init_err_sen_idx := 15;
            state1.dvar_M_HardwareMap := elit_init_error;

            state0 := state1;
        END_IF;
    END_IF;

    // Event "tau".
    IF NOT progress THEN
        b1 := (state0.dvar_M_HardwareMap) = (elit_init_sensor_check);
        b1 := b1 AND (NOT(ivar_s_pusher3_in));
        IF b1 THEN
            progress := TRUE;
            state1 := state0;

            state1.dvar_M_HardwareMap_init_err_sen_idx := 16;
            state1.dvar_M_HardwareMap := elit_init_error;

            state0 := state1;
        END_IF;
    END_IF;

    // Event "tau".
    IF NOT progress THEN
        b1 := (state0.dvar_M_HardwareMap) = (elit_init_sensor_check);
        b1 := b1 AND (ivar_s_pusher3_out);
        IF b1 THEN
            progress := TRUE;
            state1 := state0;

            state1.dvar_M_HardwareMap_init_err_sen_idx := 17;
            state1.dvar_M_HardwareMap := elit_init_error;

            state0 := state1;
        END_IF;
    END_IF;

    // Event "tau".
    IF NOT progress THEN
        b1 := (state0.dvar_M_HardwareMap) = (elit_init_sensor_check);
        b1 := b1 AND (NOT(ivar_s_stack3filled));
        IF b1 THEN
            progress := TRUE;
            state1 := state0;

            state1.dvar_M_HardwareMap_init_err_sen_idx := 18;
            state1.dvar_M_HardwareMap := elit_init_error;

            state0 := state1;
        END_IF;
    END_IF;

    // Event "tau".
    IF NOT progress THEN
        b1 := (state0.dvar_M_HardwareMap) = (elit_init_sensor_check);
        b1 := b1 AND (ivar_s_product3);
        IF b1 THEN
            progress := TRUE;
            state1 := state0;

            state1.dvar_M_HardwareMap_init_err_sen_idx := 19;
            state1.dvar_M_HardwareMap := elit_init_error;

            state0 := state1;
        END_IF;
    END_IF;

    // Event "tau".
    IF NOT progress THEN
        b1 := (state0.dvar_M_HardwareMap) = (elit_init_sensor_check);
        b1 := b1 AND (ivar_s_Hstartbutton);
        IF b1 THEN
            progress := TRUE;
            state1 := state0;

            state1.dvar_M_HardwareMap_init_err_sen_idx := 22;
            state1.dvar_M_HardwareMap := elit_init_error;

            state0 := state1;
        END_IF;
    END_IF;

    // Event "tau".
    IF NOT progress THEN
        b1 := (state0.dvar_M_HardwareMap) = (elit_init_sensor_check);
        b1 := b1 AND (NOT(ivar_s_Hstopbutton));
        IF b1 THEN
            progress := TRUE;
            state1 := state0;

            state1.dvar_M_HardwareMap_init_err_sen_idx := 23;
            state1.dvar_M_HardwareMap := elit_init_error;

            state0 := state1;
        END_IF;
    END_IF;

    // Event "tau".
    IF NOT progress THEN
        b1 := (state0.dvar_M_HardwareMap) = (elit_init_sensor_check);
        b1 := b1 AND (ivar_s_Hautoswitch);
        IF b1 THEN
            progress := TRUE;
            state1 := state0;

            state1.dvar_M_HardwareMap_init_err_sen_idx := 24;
            state1.dvar_M_HardwareMap := elit_init_error;

            state0 := state1;
        END_IF;
    END_IF;

    // Event "tau".
    IF NOT progress THEN
        b1 := (state0.dvar_M_HardwareMap) = (elit_init_sensor_check);
        b1 := b1 AND (ivar_s_Hresetbutton);
        IF b1 THEN
            progress := TRUE;
            state1 := state0;

            state1.dvar_M_HardwareMap_init_err_sen_idx := 25;
            state1.dvar_M_HardwareMap := elit_init_error;

            state0 := state1;
        END_IF;
    END_IF;

    // Event "tau".
    IF NOT progress THEN
        b1 := (state0.dvar_M_HardwareMap) = (elit_init_sensor_check);
        b1 := b1 AND (ivar_s_Hin4);
        IF b1 THEN
            progress := TRUE;
            state1 := state0;

            state1.dvar_M_HardwareMap_init_err_sen_idx := 26;
            state1.dvar_M_HardwareMap := elit_init_error;

            state0 := state1;
        END_IF;
    END_IF;

    // Event "tau".
    IF NOT progress THEN
        b1 := (state0.dvar_M_HardwareMap) = (elit_init_sensor_check);
        b1 := b1 AND (ivar_s_Hin5);
        IF b1 THEN
            progress := TRUE;
            state1 := state0;

            state1.dvar_M_HardwareMap_init_err_sen_idx := 27;
            state1.dvar_M_HardwareMap := elit_init_error;

            state0 := state1;
        END_IF;
    END_IF;

    // Event "tau".
    IF NOT progress THEN
        b1 := (state0.dvar_M_HardwareMap) = (elit_init_sensor_check);
        b1 := b1 AND (ivar_s_Hin6);
        IF b1 THEN
            progress := TRUE;
            state1 := state0;

            state1.dvar_M_HardwareMap_init_err_sen_idx := 28;
            state1.dvar_M_HardwareMap := elit_init_error;

            state0 := state1;
        END_IF;
    END_IF;

    // Event "tau".
    IF NOT progress THEN
        b1 := (state0.dvar_M_HardwareMap) = (elit_init_sensor_check);
        b1 := b1 AND (ivar_s_Hin7);
        IF b1 THEN
            progress := TRUE;
            state1 := state0;

            state1.dvar_M_HardwareMap_init_err_sen_idx := 29;
            state1.dvar_M_HardwareMap := elit_init_error;

            state0 := state1;
        END_IF;
    END_IF;

    // Event "tau".
    IF NOT progress THEN
        b1 := (state0.dvar_M_HardwareMap) = (elit_init_sensor_check);
        b1 := b1 AND (ivar_s_xpos_at1);
        IF b1 THEN
            progress := TRUE;
            state1 := state0;

            state1.dvar_M_HardwareMap_init_err_sen_idx := 33;
            state1.dvar_M_HardwareMap := elit_init_error;

            state0 := state1;
        END_IF;
    END_IF;

    // Event "tau".
    IF NOT progress THEN
        b1 := (state0.dvar_M_HardwareMap) = (elit_init_sensor_check);
        b1 := b1 AND (ivar_s_xpos_at2);
        IF b1 THEN
            progress := TRUE;
            state1 := state0;

            state1.dvar_M_HardwareMap_init_err_sen_idx := 34;
            state1.dvar_M_HardwareMap := elit_init_error;

            state0 := state1;
        END_IF;
    END_IF;

    // Event "tau".
    IF NOT progress THEN
        b1 := (state0.dvar_M_HardwareMap) = (elit_init_sensor_check);
        b1 := b1 AND (ivar_s_xpos_at3);
        IF b1 THEN
            progress := TRUE;
            state1 := state0;

            state1.dvar_M_HardwareMap_init_err_sen_idx := 35;
            state1.dvar_M_HardwareMap := elit_init_error;

            state0 := state1;
        END_IF;
    END_IF;

    // Event "tau".
    IF NOT progress THEN
        b1 := (state0.dvar_M_HardwareMap) = (elit_init_sensor_check);
        b1 := b1 AND (NOT(ivar_s_xpos_atdrop));
        IF b1 THEN
            progress := TRUE;
            state1 := state0;

            state1.dvar_M_HardwareMap_init_err_sen_idx := 36;
            state1.dvar_M_HardwareMap := elit_init_error;

            state0 := state1;
        END_IF;
    END_IF;

    // Event "tau".
    IF NOT progress THEN
        b1 := (state0.dvar_M_HardwareMap) = (elit_init_sensor_check);
        b1 := b1 AND (NOT(ivar_s_zpos_atup));
        IF b1 THEN
            progress := TRUE;
            state1 := state0;

            state1.dvar_M_HardwareMap_init_err_sen_idx := 37;
            state1.dvar_M_HardwareMap := elit_init_error;

            state0 := state1;
        END_IF;
    END_IF;

    // Event "tau".
    IF NOT progress THEN
        b1 := (state0.dvar_M_HardwareMap) = (elit_init_sensor_check);
        b1 := b1 AND (ivar_s_zpos_atdown);
        IF b1 THEN
            progress := TRUE;
            state1 := state0;

            state1.dvar_M_HardwareMap_init_err_sen_idx := 38;
            state1.dvar_M_HardwareMap := elit_init_error;

            state0 := state1;
        END_IF;
    END_IF;

    // Event "tau".
    IF NOT progress THEN
        b1 := (state0.dvar_M_HardwareMap) = (elit_init_sensor_check);
        b1 := b1 AND (ivar_s_gripper);
        IF b1 THEN
            progress := TRUE;
            state1 := state0;

            state1.dvar_M_HardwareMap_init_err_sen_idx := 39;
            state1.dvar_M_HardwareMap := elit_init_error;

            state0 := state1;
        END_IF;
    END_IF;

    // Event "tau".
    IF NOT progress THEN
        b1 := (state0.dvar_M_HardwareMap) = (elit_init_sensor_check);
        b1 := b1 AND (ivar_s_transfer_atpickup);
        IF b1 THEN
            progress := TRUE;
            state1 := state0;

            state1.dvar_M_HardwareMap_init_err_sen_idx := 40;
            state1.dvar_M_HardwareMap := elit_init_error;

            state0 := state1;
        END_IF;
    END_IF;

    // Event "tau".
    IF NOT progress THEN
        b1 := (state0.dvar_M_HardwareMap) = (elit_init_sensor_check);
        b1 := b1 AND (ivar_s_transfer_atdrop);
        IF b1 THEN
            progress := TRUE;
            state1 := state0;

            state1.dvar_M_HardwareMap_init_err_sen_idx := 41;
            state1.dvar_M_HardwareMap := elit_init_error;

            state0 := state1;
        END_IF;
    END_IF;

    // Event "tau".
    IF NOT progress THEN
        b1 := (state0.dvar_M_HardwareMap) = (elit_init_sensor_check);
        b1 := b1 AND (NOT(ivar_s_transfer_athalfway));
        IF b1 THEN
            progress := TRUE;
            state1 := state0;

            state1.dvar_M_HardwareMap_init_err_sen_idx := 42;
            state1.dvar_M_HardwareMap := elit_init_error;

            state0 := state1;
        END_IF;
    END_IF;

    // Event "tau".
    IF NOT progress THEN
        b1 := (state0.dvar_M_HardwareMap) = (elit_init_sensor_check);
        b1 := b1 AND (ivar_s_vacuum);
        IF b1 THEN
            progress := TRUE;
            state1 := state0;

            state1.dvar_M_HardwareMap_init_err_sen_idx := 43;
            state1.dvar_M_HardwareMap := elit_init_error;

            state0 := state1;
        END_IF;
    END_IF;

    // Event "tau".
    IF NOT progress THEN
        b1 := (state0.dvar_M_HardwareMap) = (elit_init_sensor_check);
        b1 := b1 AND (ivar_s_product4);
        IF b1 THEN
            progress := TRUE;
            state1 := state0;

            state1.dvar_M_HardwareMap_init_err_sen_idx := 44;
            state1.dvar_M_HardwareMap := elit_init_error;

            state0 := state1;
        END_IF;
    END_IF;

    // Event "tau".
    IF NOT progress THEN
        b1 := (state0.dvar_M_HardwareMap) = (elit_init_sensor_check);
        b1 := b1 AND (NOT(ivar_s_Dstartbutton));
        b1 := b1 AND (ivar_s_Dstopbutton);
        b1 := b1 AND (NOT(ivar_s_Dautoswitch));
        b1 := b1 AND (NOT(ivar_s_Dresetbutton));
        b1 := b1 AND (NOT(ivar_s_Din4));
        b1 := b1 AND (NOT(ivar_s_Din5));
        b1 := b1 AND (NOT(ivar_s_Din6));
        b1 := b1 AND (NOT(ivar_s_Din7));
        b1 := b1 AND (ivar_s_pusher1_in);
        b1 := b1 AND (NOT(ivar_s_pusher1_out));
        b1 := b1 AND (ivar_s_stack1filled);
        b1 := b1 AND (NOT(ivar_s_product1));
        b1 := b1 AND (ivar_s_pusher2_in);
        b1 := b1 AND (NOT(ivar_s_pusher2_out));
        b1 := b1 AND (ivar_s_stack2filled);
        b1 := b1 AND (NOT(ivar_s_product2));
        b1 := b1 AND (ivar_s_pusher3_in);
        b1 := b1 AND (NOT(ivar_s_pusher3_out));
        b1 := b1 AND (ivar_s_stack3filled);
        b1 := b1 AND (NOT(ivar_s_product3));
        b1 := b1 AND (NOT(ivar_s_Hstartbutton));
        b1 := b1 AND (ivar_s_Hstopbutton);
        b1 := b1 AND (NOT(ivar_s_Hautoswitch));
        b1 := b1 AND (NOT(ivar_s_Hresetbutton));
        b1 := b1 AND (NOT(ivar_s_Hin4));
        b1 := b1 AND (NOT(ivar_s_Hin5));
        b1 := b1 AND (NOT(ivar_s_Hin6));
        b1 := b1 AND (NOT(ivar_s_Hin7));
        b1 := b1 AND (NOT(ivar_s_xpos_at1));
        b1 := b1 AND (NOT(ivar_s_xpos_at2));
        b1 := b1 AND (NOT(ivar_s_xpos_at3));
        b1 := b1 AND (ivar_s_xpos_atdrop);
        b1 := b1 AND (ivar_s_zpos_atup);
        b1 := b1 AND (NOT(ivar_s_zpos_atdown));
        b1 := b1 AND (NOT(ivar_s_gripper));
        b1 := b1 AND (NOT(ivar_s_transfer_atpickup));
        b1 := b1 AND (NOT(ivar_s_transfer_atdrop));
        b1 := b1 AND (ivar_s_transfer_athalfway);
        b1 := b1 AND (NOT(ivar_s_vacuum));
        b1 := b1 AND (NOT(ivar_s_product4));
        IF b1 THEN
            progress := TRUE;
            state1 := state0;

            state1.dvar_M_HardwareMap := elit_init_ok;

            state0 := state1;
        END_IF;
    END_IF;

    // Event "tau".
    IF NOT progress THEN
        b1 := (state0.dvar_M_HardwareMap) = (elit_init_error);
        b1 := b1 AND ((state0.cvar_M_HardwareMap_t) >= (0.5));
        b1 := b1 AND ((state0.dvar_M_HardwareMap_init_err_led_idx) = (0));
        IF b1 THEN
            progress := TRUE;
            state1 := state0;

            state1.cvar_M_HardwareMap_t := 0.0;
            state1.dvar_M_HardwareMap_init_err_led_idx := 1;
            state1.dvar_M_HardwareMap_out_a_DledQ1 := TRUE;
            state1.dvar_M_HardwareMap_out_a_DledQ2 := FALSE;
            state1.dvar_M_HardwareMap_out_a_HledQ1 := TRUE;
            state1.dvar_M_HardwareMap_out_a_HledQ2 := FALSE;

            state0 := state1;
        END_IF;
    END_IF;

    // Event "tau".
    IF NOT progress THEN
        b1 := (state0.dvar_M_HardwareMap) = (elit_init_error);
        b1 := b1 AND ((state0.cvar_M_HardwareMap_t) >= (0.5));
        b1 := b1 AND ((state0.dvar_M_HardwareMap_init_err_led_idx) = (1));
        IF b1 THEN
            progress := TRUE;
            state1 := state0;

            state1.cvar_M_HardwareMap_t := 0.0;
            state1.dvar_M_HardwareMap_init_err_led_idx := 0;
            state1.dvar_M_HardwareMap_out_a_DledQ1 := FALSE;
            state1.dvar_M_HardwareMap_out_a_DledQ2 := TRUE;
            state1.dvar_M_HardwareMap_out_a_HledQ1 := FALSE;
            state1.dvar_M_HardwareMap_out_a_HledQ2 := TRUE;

            state0 := state1;
        END_IF;
    END_IF;

    // Event "tau".
    IF NOT progress THEN
        IF (state0.dvar_M_HardwareMap) = (elit_init_ok) THEN
            progress := TRUE;
            state1 := state0;

            state1.dvar_M_HardwareMap_out_a_DledQ1 := FALSE;
            state1.dvar_M_HardwareMap_out_a_DledQ2 := FALSE;
            state1.dvar_M_HardwareMap_out_a_HledQ1 := FALSE;
            state1.dvar_M_HardwareMap_out_a_HledQ2 := FALSE;
            state1.dvar_M_HardwareMap := elit_initialized;

            state0 := state1;
        END_IF;
    END_IF;

    // Event "tau".
    IF NOT progress THEN
        b1 := (state0.dvar_M_HardwareMap) = (elit_initialized);
        b1 := b1 AND ((state0.dvar_M_HardwareMap_out_a_Dstartled) <> (alg_a_Dstartled(state0)));
        IF b1 THEN
            progress := TRUE;
            state1 := state0;

            state1.dvar_M_HardwareMap_out_a_Dstartled := alg_a_Dstartled(state0);

            state0 := state1;
        END_IF;
    END_IF;

    // Event "tau".
    IF NOT progress THEN
        b1 := (state0.dvar_M_HardwareMap) = (elit_initialized);
        b1 := b1 AND ((state0.dvar_M_HardwareMap_out_a_Dresetled) <> (alg_a_Dresetled(state0)));
        IF b1 THEN
            progress := TRUE;
            state1 := state0;

            state1.dvar_M_HardwareMap_out_a_Dresetled := alg_a_Dresetled(state0);

            state0 := state1;
        END_IF;
    END_IF;

    // Event "tau".
    IF NOT progress THEN
        b1 := (state0.dvar_M_HardwareMap) = (elit_initialized);
        b1 := b1 AND ((state0.dvar_M_HardwareMap_out_a_DledQ1) <> (FALSE));
        IF b1 THEN
            progress := TRUE;
            state1 := state0;

            state1.dvar_M_HardwareMap_out_a_DledQ1 := FALSE;

            state0 := state1;
        END_IF;
    END_IF;

    // Event "tau".
    IF NOT progress THEN
        b1 := (state0.dvar_M_HardwareMap) = (elit_initialized);
        b1 := b1 AND ((state0.dvar_M_HardwareMap_out_a_DledQ2) <> (FALSE));
        IF b1 THEN
            progress := TRUE;
            state1 := state0;

            state1.dvar_M_HardwareMap_out_a_DledQ2 := FALSE;

            state0 := state1;
        END_IF;
    END_IF;

    // Event "tau".
    IF NOT progress THEN
        b1 := (state0.dvar_M_HardwareMap) = (elit_initialized);
        b1 := b1 AND ((state0.dvar_M_HardwareMap_out_a_Dout4) <> (ivar_a_Dout4));
        IF b1 THEN
            progress := TRUE;
            state1 := state0;

            state1.dvar_M_HardwareMap_out_a_Dout4 := ivar_a_Dout4;

            state0 := state1;
        END_IF;
    END_IF;

    // Event "tau".
    IF NOT progress THEN
        b1 := (state0.dvar_M_HardwareMap) = (elit_initialized);
        b1 := b1 AND ((state0.dvar_M_HardwareMap_out_a_Dout5) <> (ivar_a_Dout5));
        IF b1 THEN
            progress := TRUE;
            state1 := state0;

            state1.dvar_M_HardwareMap_out_a_Dout5 := ivar_a_Dout5;

            state0 := state1;
        END_IF;
    END_IF;

    // Event "tau".
    IF NOT progress THEN
        b1 := (state0.dvar_M_HardwareMap) = (elit_initialized);
        b1 := b1 AND ((state0.dvar_M_HardwareMap_out_a_Dout6) <> (ivar_a_Dout6));
        IF b1 THEN
            progress := TRUE;
            state1 := state0;

            state1.dvar_M_HardwareMap_out_a_Dout6 := ivar_a_Dout6;

            state0 := state1;
        END_IF;
    END_IF;

    // Event "tau".
    IF NOT progress THEN
        b1 := (state0.dvar_M_HardwareMap) = (elit_initialized);
        b1 := b1 AND ((state0.dvar_M_HardwareMap_out_a_Dout7) <> (ivar_a_Dout7));
        IF b1 THEN
            progress := TRUE;
            state1 := state0;

            state1.dvar_M_HardwareMap_out_a_Dout7 := ivar_a_Dout7;

            state0 := state1;
        END_IF;
    END_IF;

    // Event "tau".
    IF NOT progress THEN
        b1 := (state0.dvar_M_HardwareMap) = (elit_initialized);
        b1 := b1 AND ((state0.dvar_M_HardwareMap_out_a_pusher1) <> (alg_a_pusher1(state0)));
        IF b1 THEN
            progress := TRUE;
            state1 := state0;

            state1.dvar_M_HardwareMap_out_a_pusher1 := alg_a_pusher1(state0);

            state0 := state1;
        END_IF;
    END_IF;

    // Event "tau".
    IF NOT progress THEN
        b1 := (state0.dvar_M_HardwareMap) = (elit_initialized);
        b1 := b1 AND ((state0.dvar_M_HardwareMap_out_a_pusher2) <> (alg_a_pusher2(state0)));
        IF b1 THEN
            progress := TRUE;
            state1 := state0;

            state1.dvar_M_HardwareMap_out_a_pusher2 := alg_a_pusher2(state0);

            state0 := state1;
        END_IF;
    END_IF;

    // Event "tau".
    IF NOT progress THEN
        b1 := (state0.dvar_M_HardwareMap) = (elit_initialized);
        b1 := b1 AND ((state0.dvar_M_HardwareMap_out_a_pusher3) <> (alg_a_pusher3(state0)));
        IF b1 THEN
            progress := TRUE;
            state1 := state0;

            state1.dvar_M_HardwareMap_out_a_pusher3 := alg_a_pusher3(state0);

            state0 := state1;
        END_IF;
    END_IF;

    // Event "tau".
    IF NOT progress THEN
        b1 := (state0.dvar_M_HardwareMap) = (elit_initialized);
        b1 := b1 AND ((state0.dvar_M_HardwareMap_out_a_Hstartled) <> (FALSE));
        IF b1 THEN
            progress := TRUE;
            state1 := state0;

            state1.dvar_M_HardwareMap_out_a_Hstartled := FALSE;

            state0 := state1;
        END_IF;
    END_IF;

    // Event "tau".
    IF NOT progress THEN
        b1 := (state0.dvar_M_HardwareMap) = (elit_initialized);
        b1 := b1 AND ((state0.dvar_M_HardwareMap_out_a_Hresetled) <> (FALSE));
        IF b1 THEN
            progress := TRUE;
            state1 := state0;

            state1.dvar_M_HardwareMap_out_a_Hresetled := FALSE;

            state0 := state1;
        END_IF;
    END_IF;

    // Event "tau".
    IF NOT progress THEN
        b1 := (state0.dvar_M_HardwareMap) = (elit_initialized);
        b1 := b1 AND ((state0.dvar_M_HardwareMap_out_a_HledQ1) <> (FALSE));
        IF b1 THEN
            progress := TRUE;
            state1 := state0;

            state1.dvar_M_HardwareMap_out_a_HledQ1 := FALSE;

            state0 := state1;
        END_IF;
    END_IF;

    // Event "tau".
    IF NOT progress THEN
        b1 := (state0.dvar_M_HardwareMap) = (elit_initialized);
        b1 := b1 AND ((state0.dvar_M_HardwareMap_out_a_HledQ2) <> (FALSE));
        IF b1 THEN
            progress := TRUE;
            state1 := state0;

            state1.dvar_M_HardwareMap_out_a_HledQ2 := FALSE;

            state0 := state1;
        END_IF;
    END_IF;

    // Event "tau".
    IF NOT progress THEN
        b1 := (state0.dvar_M_HardwareMap) = (elit_initialized);
        b1 := b1 AND ((state0.dvar_M_HardwareMap_out_a_Hout4) <> (ivar_a_Hout4));
        IF b1 THEN
            progress := TRUE;
            state1 := state0;

            state1.dvar_M_HardwareMap_out_a_Hout4 := ivar_a_Hout4;

            state0 := state1;
        END_IF;
    END_IF;

    // Event "tau".
    IF NOT progress THEN
        b1 := (state0.dvar_M_HardwareMap) = (elit_initialized);
        b1 := b1 AND ((state0.dvar_M_HardwareMap_out_a_Hout5) <> (ivar_a_Hout5));
        IF b1 THEN
            progress := TRUE;
            state1 := state0;

            state1.dvar_M_HardwareMap_out_a_Hout5 := ivar_a_Hout5;

            state0 := state1;
        END_IF;
    END_IF;

    // Event "tau".
    IF NOT progress THEN
        b1 := (state0.dvar_M_HardwareMap) = (elit_initialized);
        b1 := b1 AND ((state0.dvar_M_HardwareMap_out_a_Hout6) <> (ivar_a_Hout6));
        IF b1 THEN
            progress := TRUE;
            state1 := state0;

            state1.dvar_M_HardwareMap_out_a_Hout6 := ivar_a_Hout6;

            state0 := state1;
        END_IF;
    END_IF;

    // Event "tau".
    IF NOT progress THEN
        b1 := (state0.dvar_M_HardwareMap) = (elit_initialized);
        b1 := b1 AND ((state0.dvar_M_HardwareMap_out_a_Hout7) <> (ivar_a_Hout7));
        IF b1 THEN
            progress := TRUE;
            state1 := state0;

            state1.dvar_M_HardwareMap_out_a_Hout7 := ivar_a_Hout7;

            state0 := state1;
        END_IF;
    END_IF;

    // Event "tau".
    IF NOT progress THEN
        b1 := (state0.dvar_M_HardwareMap) = (elit_initialized);
        b1 := b1 AND ((state0.dvar_M_HardwareMap_out_a_x2distributing) <> (alg_a_x2distributing(state0)));
        IF b1 THEN
            progress := TRUE;
            state1 := state0;

            state1.dvar_M_HardwareMap_out_a_x2distributing := alg_a_x2distributing(state0);

            state0 := state1;
        END_IF;
    END_IF;

    // Event "tau".
    IF NOT progress THEN
        b1 := (state0.dvar_M_HardwareMap) = (elit_initialized);
        b1 := b1 AND ((state0.dvar_M_HardwareMap_out_a_x2testing) <> (alg_a_x2testing(state0)));
        IF b1 THEN
            progress := TRUE;
            state1 := state0;

            state1.dvar_M_HardwareMap_out_a_x2testing := alg_a_x2testing(state0);

            state0 := state1;
        END_IF;
    END_IF;

    // Event "tau".
    IF NOT progress THEN
        b1 := (state0.dvar_M_HardwareMap) = (elit_initialized);
        b1 := b1 AND ((state0.dvar_M_HardwareMap_out_a_zdown) <> (alg_a_zdown(state0)));
        IF b1 THEN
            progress := TRUE;
            state1 := state0;

            state1.dvar_M_HardwareMap_out_a_zdown := alg_a_zdown(state0);

            state0 := state1;
        END_IF;
    END_IF;

    // Event "tau".
    IF NOT progress THEN
        b1 := (state0.dvar_M_HardwareMap) = (elit_initialized);
        b1 := b1 AND ((state0.dvar_M_HardwareMap_out_a_gripperclose) <> (alg_a_gripperclose(state0)));
        IF b1 THEN
            progress := TRUE;
            state1 := state0;

            state1.dvar_M_HardwareMap_out_a_gripperclose := alg_a_gripperclose(state0);

            state0 := state1;
        END_IF;
    END_IF;

    // Event "tau".
    IF NOT progress THEN
        b1 := (state0.dvar_M_HardwareMap) = (elit_initialized);
        b1 := b1 AND ((state0.dvar_M_HardwareMap_out_a_transfer2pickpos) <> (alg_a_transfer2pickpos(state0)));
        IF b1 THEN
            progress := TRUE;
            state1 := state0;

            state1.dvar_M_HardwareMap_out_a_transfer2pickpos := alg_a_transfer2pickpos(state0);

            state0 := state1;
        END_IF;
    END_IF;

    // Event "tau".
    IF NOT progress THEN
        b1 := (state0.dvar_M_HardwareMap) = (elit_initialized);
        b1 := b1 AND ((state0.dvar_M_HardwareMap_out_a_transfer2droppos) <> (alg_a_transfer2droppos(state0)));
        IF b1 THEN
            progress := TRUE;
            state1 := state0;

            state1.dvar_M_HardwareMap_out_a_transfer2droppos := alg_a_transfer2droppos(state0);

            state0 := state1;
        END_IF;
    END_IF;

    // Event "tau".
    IF NOT progress THEN
        b1 := (state0.dvar_M_HardwareMap) = (elit_initialized);
        b1 := b1 AND ((state0.dvar_M_HardwareMap_out_a_vacuum) <> (alg_a_vacuum(state0)));
        IF b1 THEN
            progress := TRUE;
            state1 := state0;

            state1.dvar_M_HardwareMap_out_a_vacuum := alg_a_vacuum(state0);

            state0 := state1;
        END_IF;
    END_IF;

    // Event "tau".
    IF NOT progress THEN
        b1 := (state0.dvar_M_HardwareMap) = (elit_initialized);
        b1 := b1 AND ((state0.dvar_M_HardwareMap_out_a_ejectpulse) <> (alg_a_ejectpulse(state0)));
        IF b1 THEN
            progress := TRUE;
            state1 := state0;

            state1.dvar_M_HardwareMap_out_a_ejectpulse := alg_a_ejectpulse(state0);

            state0 := state1;
        END_IF;
    END_IF;

    // Event "tau".
    IF NOT progress THEN
        b1 := (state0.dvar_M_HardwareMap) = (elit_initialized);
        b1 := b1 AND ((state0.dvar_M_HardwareMap_out_a_handlingready) <> (FALSE));
        IF b1 THEN
            progress := TRUE;
            state1 := state0;

            state1.dvar_M_HardwareMap_out_a_handlingready := FALSE;

            state0 := state1;
        END_IF;
    END_IF;

    // Event "tau".
    IF NOT progress THEN
        b1 := (state0.dvar_M_inventory1) = (elit_init2);
        b1 := b1 AND (alg_s_Dinitialized(state0));
        IF b1 THEN
            progress := TRUE;
            state1 := state0;

            state1.dvar_M_inventory1 := elit_wait_start;

            state0 := state1;
        END_IF;
    END_IF;

    // Event "tau".
    IF NOT progress THEN
        b1 := (state0.dvar_M_inventory1) = (elit_wait_start);
        b1 := b1 AND (ivar_s_Dstartbutton);
        IF b1 THEN
            progress := TRUE;
            state1 := state0;

            state1.dvar_M_inventory1 := elit_starting;

            state0 := state1;
        END_IF;
    END_IF;

    // Event "tau".
    IF NOT progress THEN
        b1 := (state0.dvar_M_inventory1) = (elit_stop);
        b1 := b1 AND (ivar_s_Dstartbutton);
        IF b1 THEN
            progress := TRUE;
            state1 := state0;

            state1.dvar_M_inventory1 := elit_starting;

            state0 := state1;
        END_IF;
    END_IF;

    // Event "tau".
    IF NOT progress THEN
        b1 := (state0.dvar_M_inventory1) = (elit_going);
        b1 := b1 AND (NOT(ivar_s_Dstopbutton));
        IF b1 THEN
            progress := TRUE;
            state1 := state0;

            state1.dvar_M_inventory1 := elit_stop;

            state0 := state1;
        END_IF;
    END_IF;

    // Event "tau".
    IF NOT progress THEN
        b1 := (state0.dvar_M_inventory2) = (elit_init2);
        b1 := b1 AND (alg_s_Dinitialized(state0));
        IF b1 THEN
            progress := TRUE;
            state1 := state0;

            state1.dvar_M_inventory2 := elit_wait_start;

            state0 := state1;
        END_IF;
    END_IF;

    // Event "tau".
    IF NOT progress THEN
        b1 := (state0.dvar_M_inventory2) = (elit_wait_start);
        b1 := b1 AND (ivar_s_Dstartbutton);
        IF b1 THEN
            progress := TRUE;
            state1 := state0;

            state1.dvar_M_inventory2 := elit_starting;

            state0 := state1;
        END_IF;
    END_IF;

    // Event "tau".
    IF NOT progress THEN
        b1 := (state0.dvar_M_inventory2) = (elit_stop);
        b1 := b1 AND (ivar_s_Dstartbutton);
        IF b1 THEN
            progress := TRUE;
            state1 := state0;

            state1.dvar_M_inventory2 := elit_starting;

            state0 := state1;
        END_IF;
    END_IF;

    // Event "tau".
    IF NOT progress THEN
        b1 := (state0.dvar_M_inventory2) = (elit_starting);
        b1 := b1 AND (ivar_s_pusher2_in);
        b1 := b1 AND (NOT(ivar_s_product2));
        IF b1 THEN
            progress := TRUE;
            state1 := state0;

            state1.dvar_M_inventory2_a_pusher2 := TRUE;
            state1.dvar_M_inventory2 := elit_going;

            state0 := state1;
        END_IF;
    END_IF;

    // Event "tau".
    IF NOT progress THEN
        b1 := (state0.dvar_M_inventory2) = (elit_starting);
        b1 := b1 AND (ivar_s_pusher2_out);
        b1 := b1 AND (ivar_s_stack1filled);
        b1 := b1 AND (state0.dvar_M_inventory2_a_pusher2);
        IF b1 THEN
            progress := TRUE;
            state1 := state0;

            state1.dvar_M_inventory2 := elit_going;

            state0 := state1;
        END_IF;
    END_IF;

    // Event "tau".
    IF NOT progress THEN
        b1 := (state0.dvar_M_inventory2) = (elit_starting);
        b1 := b1 AND (NOT(ivar_s_Dstopbutton));
        IF b1 THEN
            progress := TRUE;
            state1 := state0;

            state1.dvar_M_inventory2_a_pusher2 := FALSE;
            state1.dvar_M_inventory2 := elit_stop;

            state0 := state1;
        END_IF;
    END_IF;

    // Event "tau".
    IF NOT progress THEN
        b1 := (state0.dvar_M_inventory2) = (elit_going);
        b1 := b1 AND (ivar_s_pusher2_out);
        b1 := b1 AND (ivar_s_stack2filled);
        IF b1 THEN
            progress := TRUE;
            state1 := state0;

            state1.dvar_M_inventory2_a_pusher2 := FALSE;
            state1.dvar_M_inventory2 := elit_starting;

            state0 := state1;
        END_IF;
    END_IF;

    // Event "tau".
    IF NOT progress THEN
        b1 := (state0.dvar_M_inventory2) = (elit_going);
        b1 := b1 AND (NOT(ivar_s_Dstopbutton));
        IF b1 THEN
            progress := TRUE;
            state1 := state0;

            state1.dvar_M_inventory2 := elit_stop;

            state0 := state1;
        END_IF;
    END_IF;

    // Event "tau".
    IF NOT progress THEN
        b1 := (state0.dvar_M_inventory3) = (elit_init2);
        b1 := b1 AND (alg_s_Dinitialized(state0));
        IF b1 THEN
            progress := TRUE;
            state1 := state0;

            state1.dvar_M_inventory3 := elit_wait_start;

            state0 := state1;
        END_IF;
    END_IF;

    // Event "tau".
    IF NOT progress THEN
        b1 := (state0.dvar_M_inventory3) = (elit_wait_start);
        b1 := b1 AND (ivar_s_Dstartbutton);
        IF b1 THEN
            progress := TRUE;
            state1 := state0;

            state1.dvar_M_inventory3 := elit_starting;

            state0 := state1;
        END_IF;
    END_IF;

    // Event "tau".
    IF NOT progress THEN
        b1 := (state0.dvar_M_inventory3) = (elit_stop);
        b1 := b1 AND (ivar_s_Dstartbutton);
        IF b1 THEN
            progress := TRUE;
            state1 := state0;

            state1.dvar_M_inventory3 := elit_starting;

            state0 := state1;
        END_IF;
    END_IF;

    // Event "tau".
    IF NOT progress THEN
        b1 := (state0.dvar_M_inventory3) = (elit_starting);
        b1 := b1 AND (ivar_s_pusher3_in);
        b1 := b1 AND (NOT(ivar_s_product3));
        IF b1 THEN
            progress := TRUE;
            state1 := state0;

            state1.dvar_M_inventory3_a_pusher3 := TRUE;
            state1.dvar_M_inventory3 := elit_going;

            state0 := state1;
        END_IF;
    END_IF;

    // Event "tau".
    IF NOT progress THEN
        b1 := (state0.dvar_M_inventory3) = (elit_starting);
        b1 := b1 AND (ivar_s_pusher3_out);
        b1 := b1 AND (ivar_s_stack1filled);
        b1 := b1 AND (state0.dvar_M_inventory3_a_pusher3);
        IF b1 THEN
            progress := TRUE;
            state1 := state0;

            state1.dvar_M_inventory3 := elit_going;

            state0 := state1;
        END_IF;
    END_IF;

    // Event "tau".
    IF NOT progress THEN
        b1 := (state0.dvar_M_inventory3) = (elit_starting);
        b1 := b1 AND (NOT(ivar_s_Dstopbutton));
        IF b1 THEN
            progress := TRUE;
            state1 := state0;

            state1.dvar_M_inventory3_a_pusher3 := FALSE;
            state1.dvar_M_inventory3 := elit_stop;

            state0 := state1;
        END_IF;
    END_IF;

    // Event "tau".
    IF NOT progress THEN
        b1 := (state0.dvar_M_inventory3) = (elit_going);
        b1 := b1 AND (ivar_s_pusher3_out);
        b1 := b1 AND (ivar_s_stack3filled);
        IF b1 THEN
            progress := TRUE;
            state1 := state0;

            state1.dvar_M_inventory3_a_pusher3 := FALSE;
            state1.dvar_M_inventory3 := elit_starting;

            state0 := state1;
        END_IF;
    END_IF;

    // Event "tau".
    IF NOT progress THEN
        b1 := (state0.dvar_M_inventory3) = (elit_going);
        b1 := b1 AND (NOT(ivar_s_Dstopbutton));
        IF b1 THEN
            progress := TRUE;
            state1 := state0;

            state1.dvar_M_inventory3 := elit_stop;

            state0 := state1;
        END_IF;
    END_IF;

    // Event "tau".
    IF NOT progress THEN
        b1 := (state0.dvar_M_vacuum) = (elit_init2);
        b1 := b1 AND (alg_s_Dinitialized(state0));
        IF b1 THEN
            progress := TRUE;
            state1 := state0;

            state1.dvar_M_vacuum := elit_wait_start;

            state0 := state1;
        END_IF;
    END_IF;

    // Event "tau".
    IF NOT progress THEN
        b1 := (state0.dvar_M_vacuum) = (elit_wait_start);
        b1 := b1 AND (ivar_s_Dstartbutton);
        IF b1 THEN
            progress := TRUE;
            state1 := state0;

            state1.dvar_M_vacuum := elit_starting;

            state0 := state1;
        END_IF;
    END_IF;

    // Event "tau".
    IF NOT progress THEN
        b1 := (state0.dvar_M_vacuum) = (elit_clear_vacuum);
        b1 := b1 AND (ivar_s_transfer_atdrop);
        b1 := b1 AND (ivar_s_vacuum);
        IF b1 THEN
            progress := TRUE;
            state1 := state0;

            state1.dvar_M_vacuum_a_vacuum := FALSE;
            state1.dvar_M_vacuum_a_ejectpulse := TRUE;
            state1.dvar_M_vacuum_a_transfer2pickpos := TRUE;
            state1.dvar_M_vacuum_a_transfer2droppos := FALSE;
            state1.dvar_M_vacuum := elit_reset_button;

            state0 := state1;
        END_IF;
    END_IF;

    // Event "tau".
    IF NOT progress THEN
        b1 := (state0.dvar_M_vacuum) = (elit_clear_vacuum);
        b1 := b1 AND (ivar_s_transfer_atdrop);
        b1 := b1 AND (NOT(ivar_s_vacuum));
        IF b1 THEN
            progress := TRUE;
            state1 := state0;

            state1.dvar_M_vacuum_a_vacuum := FALSE;
            state1.dvar_M_vacuum_a_ejectpulse := FALSE;
            state1.dvar_M_vacuum_a_transfer2pickpos := TRUE;
            state1.dvar_M_vacuum_a_transfer2droppos := FALSE;
            state1.dvar_M_vacuum := elit_reset_button;

            state0 := state1;
        END_IF;
    END_IF;

    // Event "tau".
    IF NOT progress THEN
        b1 := (state0.dvar_M_vacuum) = (elit_reset_button);
        b1 := b1 AND (ivar_s_transfer_athalfway);
        IF b1 THEN
            progress := TRUE;
            state1 := state0;

            state1.dvar_M_vacuum_a_transfer2pickpos := FALSE;
            state1.dvar_M_vacuum_a_transfer2droppos := FALSE;
            state1.dvar_M_vacuum_a_ejectpulse := FALSE;
            state1.dvar_M_vacuum := elit_wait_start;

            state0 := state1;
        END_IF;
    END_IF;

    // Event "tau".
    IF NOT progress THEN
        b1 := (state0.dvar_M_vacuum) = (elit_stop);
        b1 := b1 AND (ivar_s_Dstartbutton);
        IF b1 THEN
            progress := TRUE;
            state1 := state0;

            state1.dvar_M_vacuum := elit_starting;

            state0 := state1;
        END_IF;
    END_IF;

    // Event "tau".
    IF NOT progress THEN
        b1 := (state0.dvar_M_vacuum) = (elit_stop);
        b1 := b1 AND (ivar_s_Dresetbutton);
        IF b1 THEN
            progress := TRUE;
            state1 := state0;

            state1.dvar_M_vacuum_a_transfer2droppos := TRUE;
            state1.dvar_M_vacuum_a_transfer2pickpos := FALSE;
            state1.dvar_M_vacuum := elit_clear_vacuum;

            state0 := state1;
        END_IF;
    END_IF;

    // Event "tau".
    IF NOT progress THEN
        b1 := (state0.dvar_M_vacuum) = (elit_key);
        b1 := b1 AND (NOT(ivar_s_Dautoswitch));
        IF b1 THEN
            progress := TRUE;
            state1 := state0;

            state1.dvar_M_vacuum := elit_starting;

            state0 := state1;
        END_IF;
    END_IF;

    // Event "tau".
    IF NOT progress THEN
        b1 := (state0.dvar_M_vacuum) = (elit_starting);
        b1 := b1 AND (ivar_s_Dresetbutton);
        IF b1 THEN
            progress := TRUE;
            state1 := state0;

            state1.dvar_M_vacuum_a_transfer2droppos := TRUE;
            state1.dvar_M_vacuum_a_transfer2pickpos := FALSE;
            state1.dvar_M_vacuum := elit_clear_vacuum;

            state0 := state1;
        END_IF;
    END_IF;

    // Event "tau".
    IF NOT progress THEN
        b1 := (state0.dvar_M_vacuum) = (elit_starting);
        b1 := b1 AND (NOT(ivar_s_Dstopbutton));
        IF b1 THEN
            progress := TRUE;
            state1 := state0;

            state1.dvar_M_vacuum_a_transfer2pickpos := FALSE;
            state1.dvar_M_vacuum_a_transfer2droppos := FALSE;
            state1.dvar_M_vacuum_a_ejectpulse := FALSE;
            state1.dvar_M_vacuum := elit_stop;

            state0 := state1;
        END_IF;
    END_IF;

    // Event "tau".
    IF NOT progress THEN
        b1 := (state0.dvar_M_vacuum) = (elit_starting);
        b1 := b1 AND (ivar_s_product4);
        b1 := b1 AND (ivar_s_zpos_atup);
        b1 := b1 AND (NOT(ivar_s_vacuum));
        IF b1 THEN
            progress := TRUE;
            state1 := state0;

            state1.dvar_M_vacuum_a_transfer2pickpos := TRUE;
            state1.dvar_M_vacuum := elit_pickupvac;

            state0 := state1;
        END_IF;
    END_IF;

    // Event "tau".
    IF NOT progress THEN
        b1 := (state0.dvar_M_vacuum) = (elit_starting);
        b1 := b1 AND (ivar_s_vacuum);
        IF b1 THEN
            progress := TRUE;
            state1 := state0;

            state1.dvar_M_vacuum_a_transfer2droppos := TRUE;
            state1.dvar_M_vacuum := elit_pickupvac;

            state0 := state1;
        END_IF;
    END_IF;

    // Event "tau".
    IF NOT progress THEN
        b1 := (state0.dvar_M_vacuum) = (elit_starting);
        b1 := b1 AND (ivar_s_transfer_athalfway);
        b1 := b1 AND (ivar_s_Dautoswitch);
        b1 := b1 AND (NOT(ivar_s_vacuum));
        IF b1 THEN
            progress := TRUE;
            state1 := state0;

            state1.dvar_M_vacuum_a_transfer2pickpos := FALSE;
            state1.dvar_M_vacuum_a_transfer2droppos := FALSE;
            state1.dvar_M_vacuum_a_ejectpulse := FALSE;
            state1.dvar_M_vacuum := elit_key;

            state0 := state1;
        END_IF;
    END_IF;

    // Event "tau".
    IF NOT progress THEN
        b1 := (state0.dvar_M_vacuum) = (elit_pickupvac);
        b1 := b1 AND (ivar_s_Dresetbutton);
        IF b1 THEN
            progress := TRUE;
            state1 := state0;

            state1.dvar_M_vacuum_a_transfer2droppos := TRUE;
            state1.dvar_M_vacuum_a_transfer2pickpos := FALSE;
            state1.dvar_M_vacuum := elit_clear_vacuum;

            state0 := state1;
        END_IF;
    END_IF;

    // Event "tau".
    IF NOT progress THEN
        b1 := (state0.dvar_M_vacuum) = (elit_pickupvac);
        b1 := b1 AND (NOT(ivar_s_Dstopbutton));
        IF b1 THEN
            progress := TRUE;
            state1 := state0;

            state1.dvar_M_vacuum_a_transfer2pickpos := FALSE;
            state1.dvar_M_vacuum_a_transfer2droppos := FALSE;
            state1.dvar_M_vacuum_a_ejectpulse := FALSE;
            state1.dvar_M_vacuum := elit_stop;

            state0 := state1;
        END_IF;
    END_IF;

    // Event "tau".
    IF NOT progress THEN
        b1 := (state0.dvar_M_vacuum) = (elit_pickupvac);
        b1 := b1 AND (ivar_s_transfer_atpickup);
        b1 := b1 AND (NOT(ivar_s_vacuum));
        IF b1 THEN
            progress := TRUE;
            state1 := state0;

            state1.dvar_M_vacuum_a_transfer2pickpos := FALSE;
            state1.dvar_M_vacuum_a_vacuum := TRUE;
            state1.dvar_M_vacuum := elit_testingdrop;

            state0 := state1;
        END_IF;
    END_IF;

    // Event "tau".
    IF NOT progress THEN
        b1 := (state0.dvar_M_vacuum) = (elit_pickupvac);
        b1 := b1 AND (ivar_s_transfer_atdrop);
        IF b1 THEN
            progress := TRUE;
            state1 := state0;

            state1.dvar_M_vacuum_a_vacuum := FALSE;
            state1.dvar_M_vacuum_a_ejectpulse := TRUE;
            state1.dvar_M_vacuum := elit_testingdrop;

            state0 := state1;
        END_IF;
    END_IF;

    // Event "tau".
    IF NOT progress THEN
        b1 := (state0.dvar_M_vacuum) = (elit_pickupvac);
        b1 := b1 AND (ivar_s_transfer_athalfway);
        b1 := b1 AND (ivar_s_Dautoswitch);
        b1 := b1 AND (NOT(ivar_s_vacuum));
        IF b1 THEN
            progress := TRUE;
            state1 := state0;

            state1.dvar_M_vacuum_a_transfer2pickpos := FALSE;
            state1.dvar_M_vacuum_a_transfer2droppos := FALSE;
            state1.dvar_M_vacuum_a_ejectpulse := FALSE;
            state1.dvar_M_vacuum := elit_key;

            state0 := state1;
        END_IF;
    END_IF;

    // Event "tau".
    IF NOT progress THEN
        b1 := (state0.dvar_M_vacuum) = (elit_testingdrop);
        b1 := b1 AND (ivar_s_Dresetbutton);
        IF b1 THEN
            progress := TRUE;
            state1 := state0;

            state1.dvar_M_vacuum_a_transfer2droppos := TRUE;
            state1.dvar_M_vacuum_a_transfer2pickpos := FALSE;
            state1.dvar_M_vacuum := elit_clear_vacuum;

            state0 := state1;
        END_IF;
    END_IF;

    // Event "tau".
    IF NOT progress THEN
        b1 := (state0.dvar_M_vacuum) = (elit_testingdrop);
        b1 := b1 AND (NOT(ivar_s_Dstopbutton));
        IF b1 THEN
            progress := TRUE;
            state1 := state0;

            state1.dvar_M_vacuum_a_transfer2pickpos := FALSE;
            state1.dvar_M_vacuum_a_transfer2droppos := FALSE;
            state1.dvar_M_vacuum_a_ejectpulse := FALSE;
            state1.dvar_M_vacuum := elit_stop;

            state0 := state1;
        END_IF;
    END_IF;

    // Event "tau".
    IF NOT progress THEN
        b1 := (state0.dvar_M_vacuum) = (elit_testingdrop);
        b1 := b1 AND (ivar_s_vacuum);
        b1 := b1 AND (ivar_s_transfer_atpickup);
        IF b1 THEN
            progress := TRUE;
            state1 := state0;

            state1.dvar_M_vacuum_a_transfer2droppos := TRUE;
            state1.dvar_M_vacuum := elit_starting;

            state0 := state1;
        END_IF;
    END_IF;

    // Event "tau".
    IF NOT progress THEN
        b1 := (state0.dvar_M_vacuum) = (elit_testingdrop);
        b1 := b1 AND (NOT(ivar_s_vacuum));
        b1 := b1 AND (ivar_s_transfer_atdrop);
        IF b1 THEN
            progress := TRUE;
            state1 := state0;

            state1.dvar_M_vacuum_a_transfer2pickpos := TRUE;
            state1.dvar_M_vacuum_a_transfer2droppos := FALSE;
            state1.dvar_M_vacuum := elit_rest;

            state0 := state1;
        END_IF;
    END_IF;

    // Event "tau".
    IF NOT progress THEN
        b1 := (state0.dvar_M_vacuum) = (elit_testingdrop);
        b1 := b1 AND (ivar_s_transfer_athalfway);
        b1 := b1 AND (ivar_s_Dautoswitch);
        b1 := b1 AND (NOT(ivar_s_vacuum));
        IF b1 THEN
            progress := TRUE;
            state1 := state0;

            state1.dvar_M_vacuum_a_transfer2pickpos := FALSE;
            state1.dvar_M_vacuum_a_transfer2droppos := FALSE;
            state1.dvar_M_vacuum_a_ejectpulse := FALSE;
            state1.dvar_M_vacuum := elit_key;

            state0 := state1;
        END_IF;
    END_IF;

    // Event "tau".
    IF NOT progress THEN
        b1 := (state0.dvar_M_vacuum) = (elit_rest);
        b1 := b1 AND (NOT(ivar_s_Dstopbutton));
        IF b1 THEN
            progress := TRUE;
            state1 := state0;

            state1.dvar_M_vacuum_a_transfer2pickpos := FALSE;
            state1.dvar_M_vacuum_a_transfer2droppos := FALSE;
            state1.dvar_M_vacuum_a_ejectpulse := FALSE;
            state1.dvar_M_vacuum := elit_stop;

            state0 := state1;
        END_IF;
    END_IF;

    // Event "tau".
    IF NOT progress THEN
        b1 := (state0.dvar_M_vacuum) = (elit_rest);
        b1 := b1 AND (ivar_s_transfer_athalfway);
        b1 := b1 AND (ivar_s_Dautoswitch);
        IF b1 THEN
            progress := TRUE;
            state1 := state0;

            state1.dvar_M_vacuum_a_transfer2pickpos := FALSE;
            state1.dvar_M_vacuum_a_transfer2droppos := FALSE;
            state1.dvar_M_vacuum_a_vacuum := FALSE;
            state1.dvar_M_vacuum_a_ejectpulse := FALSE;
            state1.dvar_M_vacuum := elit_key;

            state0 := state1;
        END_IF;
    END_IF;

    // Event "tau".
    IF NOT progress THEN
        b1 := (state0.dvar_M_vacuum) = (elit_rest);
        b1 := b1 AND (ivar_s_transfer_athalfway);
        b1 := b1 AND (NOT(ivar_s_Dautoswitch));
        IF b1 THEN
            progress := TRUE;
            state1 := state0;

            state1.dvar_M_vacuum_a_transfer2pickpos := FALSE;
            state1.dvar_M_vacuum_a_transfer2droppos := FALSE;
            state1.dvar_M_vacuum_a_vacuum := FALSE;
            state1.dvar_M_vacuum_a_ejectpulse := FALSE;
            state1.dvar_M_vacuum := elit_starting;

            state0 := state1;
        END_IF;
    END_IF;

    // Done with events?
    IF NOT progress THEN
        EXIT;
    END_IF;

    // Protect against events that are always enabled.
    loopCount := loopCount + 1;
    IF loopCount >= 100 THEN
        loopsKilled := loopsKilled + 1;
        EXIT;
    END_IF;
END_WHILE;

END_PROGRAM

// ---- POUs/derivcvar_M_HardwareMap_t.TcPOU
FUNCTION derivcvar_M_HardwareMap_t: LREAL
VAR_INPUT
    state: STATE;
END_VAR

derivcvar_M_HardwareMap_t := 1.0;

END_FUNCTION

// ---- POUs/alg_s_Dinitialized.TcPOU
FUNCTION alg_s_Dinitialized: BOOL
VAR_INPUT
    state: STATE;
END_VAR

alg_s_Dinitialized := (state.dvar_M_HardwareMap) = (elit_initialized);

END_FUNCTION

// ---- POUs/alg_s_Hinitialized.TcPOU
FUNCTION alg_s_Hinitialized: BOOL
VAR_INPUT
    state: STATE;
END_VAR

alg_s_Hinitialized := (state.dvar_M_HardwareMap) = (elit_initialized);

END_FUNCTION
